	16#00000FE6:
		F_EtherCAT_VendorIDtoString := 'Specter Aerospace Inc.';

	16#00000FE7:
		F_EtherCAT_VendorIDtoString := 'VITZRO VM CO., LTD.';

	16#00000FE8:
		F_EtherCAT_VendorIDtoString := 'Follow Cam Solutions';

	16#00000FE9:
		F_EtherCAT_VendorIDtoString := 'Chengdu Jixing Plasma Technology Co., Ltd.';

	16#00000FEA:
		F_EtherCAT_VendorIDtoString := 'Shenzhen WisdaTech Co., Ltd.';

	16#00000FEC:
		F_EtherCAT_VendorIDtoString := 'Li-tech AS';

	16#00000FED:
		F_EtherCAT_VendorIDtoString := 'Contour Advanced Systems BV';

	16#00000FEE:
		F_EtherCAT_VendorIDtoString := 'Camera Positioning Systems Inc';

	16#00000FEF:
		F_EtherCAT_VendorIDtoString := 'MISUMI (CHINA) PRECISION MACHINERY TRADING CO., LTD.';

	16#00000FF0:
		F_EtherCAT_VendorIDtoString := 'D-CLUE Technologies Co., Ltd.';

	16#00000FF1:
		F_EtherCAT_VendorIDtoString := 'The Board of Trustees of the University of Illinois on behalf of the University of Illinois Chicago';

	16#00000FF2:
		F_EtherCAT_VendorIDtoString := 'Texas A&M University, College of Engineering, J. Mike Walker 66 Department of Mechanical Engineering, Robotics and Automation Design Lab';

	16#00000FF3:
		F_EtherCAT_VendorIDtoString := 'Japan Minicomputer Systems Co., Ltd.';

	16#00000FF4:
		F_EtherCAT_VendorIDtoString := 'Sun Automation Co.,Ltd';

	16#00000FF5:
		F_EtherCAT_VendorIDtoString := 'Puruvesi Automation Inc.';

	16#00000FF6:
		F_EtherCAT_VendorIDtoString := 'Shenzhen Hans Focus Technology Co., Ltd.';

	16#00000FF8:
		F_EtherCAT_VendorIDtoString := 'TAIWAN CHELIC Co., Ltd.';

	16#00000FF9:
		F_EtherCAT_VendorIDtoString := 'RoboDesign Co.,Ltd.';

	16#00000FFA:
		F_EtherCAT_VendorIDtoString := 'PineSolution Co., Ltd.';

	16#00000FFB:
		F_EtherCAT_VendorIDtoString := 'Hangzhou Fisun Intelligency & Technology Co., Ltd.';

	16#00000FFC:
		F_EtherCAT_VendorIDtoString := 'A&D Technology, Inc.';

	16#00000FFD:
		F_EtherCAT_VendorIDtoString := 'IDEC CORPORATION';

	16#00000FFE:
		F_EtherCAT_VendorIDtoString := 'Atel Corp.';

	16#00000FFF:
		F_EtherCAT_VendorIDtoString := 'ZEROSYSTEM CO,LTD';

	16#00001000:
		F_EtherCAT_VendorIDtoString := 'Motiv Robotics, Inc.';

	16#00001001:
		F_EtherCAT_VendorIDtoString := 'Ray-Links (Beijing) Technologies Co., Ltd.';

	16#00001002:
		F_EtherCAT_VendorIDtoString := 'Centro de Automatica y Robotica UPM-CSIC';

	16#00001003:
		F_EtherCAT_VendorIDtoString := 'PLAYTG Co., Ltd.';

	16#00001004:
		F_EtherCAT_VendorIDtoString := 'Shenzhen Huaxin Semiconductor Equipment Technology Co., Ltd.';

	16#00001005:
		F_EtherCAT_VendorIDtoString := 'LT Global Trade Limited dba Eco-Drive Max';

	16#00001006:
		F_EtherCAT_VendorIDtoString := 'SiGaN AG';

	16#00001007:
		F_EtherCAT_VendorIDtoString := 'MOTOREVO ROBOTICS CO.,LTD.';

	16#00001008:
		F_EtherCAT_VendorIDtoString := 'Rheinmetall Canada Inc.';

	16#00001009:
		F_EtherCAT_VendorIDtoString := 'Smart Buildings BVBA';

	16#0000100A:
		F_EtherCAT_VendorIDtoString := 'AixControl GmbH';

	16#0000100B:
		F_EtherCAT_VendorIDtoString := 'Lumina Power, Inc.';

	16#0000100C:
		F_EtherCAT_VendorIDtoString := 'Cryosol-World bv';

	16#0000100D:
		F_EtherCAT_VendorIDtoString := 'Aitoly Instruments Co., Ltd';

	16#0000100E:
		F_EtherCAT_VendorIDtoString := 'FUTUREWORKS';

	16#0000100F:
		F_EtherCAT_VendorIDtoString := 'Changsha University of Science & Technology, School of Physics & Electronic Science';

	16#00001010:
		F_EtherCAT_VendorIDtoString := 'NEXTW Technology CO., LTD.';

	16#00001011:
		F_EtherCAT_VendorIDtoString := 'H4 Inc.';

	16#00001012:
		F_EtherCAT_VendorIDtoString := 'ZHEJIANG SUPCON INFORMATION CO.,LTD.';

	16#00001013:
		F_EtherCAT_VendorIDtoString := 'oKSitem Otomasyon Ltd. Sti.';

	16#00001014:
		F_EtherCAT_VendorIDtoString := 'CSIM INC.';

	16#00001015:
		F_EtherCAT_VendorIDtoString := 'Valvan NV';

	16#00001016:
		F_EtherCAT_VendorIDtoString := 'ASAHI ENGINEERING CO.,LTD.';

	16#00001017:
		F_EtherCAT_VendorIDtoString := 'Weifang Ouxin Intelligent Control Technology Co., LTD';

	16#00001018:
		F_EtherCAT_VendorIDtoString := 'GZ Photonics Technology Co., Ltd.';

	16#00001019:
		F_EtherCAT_VendorIDtoString := 'Optoscan S.r.l.';

	16#0000101A:
		F_EtherCAT_VendorIDtoString := 'Ningbo Huayuan Machinery Technology Co., Ltd.';

	16#0000101B:
		F_EtherCAT_VendorIDtoString := 'Laza Medical, Inc.';

	16#0000101C:
		F_EtherCAT_VendorIDtoString := 'Vectioneer BV';

	16#0000101D:
		F_EtherCAT_VendorIDtoString := 'Huasteigen (Ningbo) Automation Technology Co.,Ltd.';

	16#00001020:
		F_EtherCAT_VendorIDtoString := 'PDM Industrial Excellence B.V.';

	16#00001022:
		F_EtherCAT_VendorIDtoString := 'SV Sistemi di Sicurezza';

	16#00001023:
		F_EtherCAT_VendorIDtoString := 'Lynx Robotics LLC';

	16#00001024:
		F_EtherCAT_VendorIDtoString := 'Jcast Networks Korea, Inc.';

	16#00001025:
		F_EtherCAT_VendorIDtoString := 'AcroComm Corporation';

	16#00001026:
		F_EtherCAT_VendorIDtoString := 'Hacint Intelligence Technology Co., Ltd.';

	16#00001027:
		F_EtherCAT_VendorIDtoString := 'Vision Hardware Partner';

	16#00001028:
		F_EtherCAT_VendorIDtoString := 'Forbes Marshall Pvt. Ltd.';

	16#00001029:
		F_EtherCAT_VendorIDtoString := 'Shenzhen Sunvision Technology Co., Ltd.';

	16#0000102A:
		F_EtherCAT_VendorIDtoString := 'ASAP Electronics GmbH';

	16#0000102B:
		F_EtherCAT_VendorIDtoString := 'Matrox Electronic Systems Ltd.';

	16#0000102C:
		F_EtherCAT_VendorIDtoString := 'Shanghai Zhentai Instrument Co., Ltd.';

	16#0000102D:
		F_EtherCAT_VendorIDtoString := 'ROHM Co., Ltd.';

	16#0000102E:
		F_EtherCAT_VendorIDtoString := 'Chengdu SeaDee Technology Co.,Ltd.';

	16#0000102F:
		F_EtherCAT_VendorIDtoString := 'Huazhuo Measurement and Control Technology (Shenzhen) Co., Ltd.';

	16#00001030:
		F_EtherCAT_VendorIDtoString := 'Advanced Design Technology Co.,Ltd';

	16#00001031:
		F_EtherCAT_VendorIDtoString := 'MI-Partners B.V.';

	16#00001032:
		F_EtherCAT_VendorIDtoString := 'Beijing Hanwen Wangxing Technology Co., Ltd';

	16#00001033:
		F_EtherCAT_VendorIDtoString := 'nexo SrL';

	16#00001034:
		F_EtherCAT_VendorIDtoString := 'Simplex Motion AB';

	16#00001035:
		F_EtherCAT_VendorIDtoString := 'Wuxi Juxie Intelligent Drive Co.,Ltd.';

	16#00001036:
		F_EtherCAT_VendorIDtoString := 'Shenzhen Huizhong Intelligent Technology Co., Ltd';

	16#00001037:
		F_EtherCAT_VendorIDtoString := 'THEISSL systems GmbH';

	16#00001038:
		F_EtherCAT_VendorIDtoString := 'VOLAS GmbH';

	16#00001039:
		F_EtherCAT_VendorIDtoString := 'ASTI Corporation';

	16#0000103A:
		F_EtherCAT_VendorIDtoString := 'ELETTRONICA G.B. SRL';

	16#0000103B:
		F_EtherCAT_VendorIDtoString := 'VELTRU AG';

	16#0000103C:
		F_EtherCAT_VendorIDtoString := 'SEMISOL Co., Ltd.';

	16#0000103D:
		F_EtherCAT_VendorIDtoString := 'GENIWORX Co., Ltd.';

	16#0000103E:
		F_EtherCAT_VendorIDtoString := 'TUODAO (SINGAPORE) PTE. LTD.';

	16#00001041:
		F_EtherCAT_VendorIDtoString := 'SISGEO SRL';

	16#00001043:
		F_EtherCAT_VendorIDtoString := 'Oelmaier Automation GmbH';

	16#00001044:
		F_EtherCAT_VendorIDtoString := 'VISHAY ADVANCED TECHNOLOGIES LTD';

	16#00001045:
		F_EtherCAT_VendorIDtoString := 'Beyond Kinematics LLC';

	16#00001046:
		F_EtherCAT_VendorIDtoString := 'Control expertise for trading Co. LTD';

	16#00001047:
		F_EtherCAT_VendorIDtoString := 'Tujian Automation Technology (Suzhou) Co., Ltd.';

	16#00001048:
		F_EtherCAT_VendorIDtoString := 'Shibaura Machine Co., Ltd.';

	16#00001049:
		F_EtherCAT_VendorIDtoString := 'Chip Right Corporation';

	16#0000104A:
		F_EtherCAT_VendorIDtoString := 'American Superconductor Corporation';

	16#0000104B:
		F_EtherCAT_VendorIDtoString := 'Emirates Automation Pvt Ltd';

	16#0000104C:
		F_EtherCAT_VendorIDtoString := 'ERL Sensors and Automation';

	16#0000104D:
		F_EtherCAT_VendorIDtoString := 'Zhuhai Yuanshicheng Technology Co., Ltd.';

	16#0000104E:
		F_EtherCAT_VendorIDtoString := 'University of Bergamo, Department of Engineering and Applied Sciences, Mechatronics and Mechanical Dynamics Lab';

	16#0000104F:
		F_EtherCAT_VendorIDtoString := 'Maxell Frontier Co., Ltd.';

	16#00001050:
		F_EtherCAT_VendorIDtoString := 'ZENSTEM CO., LTD.';

	16#00001051:
		F_EtherCAT_VendorIDtoString := 'CONEC Elektronische Bauelemente GmbH';

	16#00001052:
		F_EtherCAT_VendorIDtoString := 'Teegarden Engineering S.r.l.';

	16#00001053:
		F_EtherCAT_VendorIDtoString := 'iFORCOM KYOEI Co., Ltd.';

	16#00001054:
		F_EtherCAT_VendorIDtoString := 'Timeback Inc. dba Reflex Robotics';

	16#00001055:
		F_EtherCAT_VendorIDtoString := 'Stryker Corporation';

	16#00001056:
		F_EtherCAT_VendorIDtoString := 'Kickmaker';

	16#00001057:
		F_EtherCAT_VendorIDtoString := 'Andar Elektromekanik Sistemler Sanayi ve Ticaret Anonim Şirketi';

	16#00001058:
		F_EtherCAT_VendorIDtoString := 'Hefei Kaiyue Semiconductor Technology Co., Ltd.';

	16#00001059:
		F_EtherCAT_VendorIDtoString := 'Clean-Lasersysteme GmbH';

	16#0000105A:
		F_EtherCAT_VendorIDtoString := 'SMACH CO., Ltd.';

	16#0000105B:
		F_EtherCAT_VendorIDtoString := 'ACD Elektronik GmbH';

	16#0000105C:
		F_EtherCAT_VendorIDtoString := 'Jiangsu Houjing Technology Co., Ltd.';

	16#0000105D:
		F_EtherCAT_VendorIDtoString := 'TACSCO Co., Ltd';

	16#0000105E:
		F_EtherCAT_VendorIDtoString := 'DGA Maitrise de linformation';

	16#0000105F:
		F_EtherCAT_VendorIDtoString := 'Dasstec B2B SRL';

	16#00001060:
		F_EtherCAT_VendorIDtoString := 'Comau S.p.A.';

	16#00001061:
		F_EtherCAT_VendorIDtoString := 'Vertiv Group Corporation';

	16#00001062:
		F_EtherCAT_VendorIDtoString := 'Insystems Inc.';

	16#00001063:
		F_EtherCAT_VendorIDtoString := 'Digital Sports Solutions LLC';

	16#00001064:
		F_EtherCAT_VendorIDtoString := 'BorgRoid Inc.';

	16#00001066:
		F_EtherCAT_VendorIDtoString := 'Shanghai ZeroOne Information Technology Co., Ltd.';

	16#00001067:
		F_EtherCAT_VendorIDtoString := 'STREAK – Engenharia em Automacao, LDA';

	16#00001068:
		F_EtherCAT_VendorIDtoString := 'Seurat Technologies, Inc.';

	16#00001069:
		F_EtherCAT_VendorIDtoString := 'EMBETTER TECHNOLOGIES PRIVATE LIMITED';

	16#0000106A:
		F_EtherCAT_VendorIDtoString := 'Beijing Regulate Technology Co., Ltd.';

	16#0000106B:
		F_EtherCAT_VendorIDtoString := 'Electronics Corporation of India Ltd.';

	16#0000106C:
		F_EtherCAT_VendorIDtoString := 'Cargt, Inc';

	16#0000106D:
		F_EtherCAT_VendorIDtoString := 'Shanghai Paipin Optoelectronic Technology Co., Ltd.';

	16#0000106E:
		F_EtherCAT_VendorIDtoString := 'Coherent Switzerland AG';

	16#0000106F:
		F_EtherCAT_VendorIDtoString := 'IP CAMP Limited Liability Company';

	16#00001071:
		F_EtherCAT_VendorIDtoString := 'Suzhou Ouluda Intelligent Technology Co., Ltd.';

	16#00001073:
		F_EtherCAT_VendorIDtoString := 'K&S Advanced Systems LTD';

	16#00001074:
		F_EtherCAT_VendorIDtoString := 'Roche Diagnostics GmbH';

	16#00001075:
		F_EtherCAT_VendorIDtoString := 'FerRobotics Compliant Robot Technology GmbH';

	16#00001077:
		F_EtherCAT_VendorIDtoString := 'TOKY ELECTRICAL CO., LTD.';

	16#00001078:
		F_EtherCAT_VendorIDtoString := 'ET Systems Engineering d.o.o.';

	16#00001079:
		F_EtherCAT_VendorIDtoString := 'Electrovia Technologies Corp';

	16#0000107A:
		F_EtherCAT_VendorIDtoString := 'Imperix Ltd.';

	16#0000107B:
		F_EtherCAT_VendorIDtoString := 'FoodJet B.V.';

	16#0000107C:
		F_EtherCAT_VendorIDtoString := 'Meridian Laboratory, Inc.';

	16#0000107D:
		F_EtherCAT_VendorIDtoString := 'ITECH ELECTRONIC CO., LTD.';

	16#0000107E:
		F_EtherCAT_VendorIDtoString := 'DANNIE ELEKTRONİK VE ELEKTRİK LTD.';

	16#0000107F:
		F_EtherCAT_VendorIDtoString := 'logi.cals GmbH';

	16#00001080:
		F_EtherCAT_VendorIDtoString := 'Unionx (Wuhan) Industrial Technology Co., Ltd.';

	16#00001081:
		F_EtherCAT_VendorIDtoString := 'Shenzhen ASunDar Electronics Co., Ltd.';

	16#00001082:
		F_EtherCAT_VendorIDtoString := 'Artesyn Embedded Technologies Philippines Inc.';

	16#00001083:
		F_EtherCAT_VendorIDtoString := 'Wuxi Dixin Technology Co., Ltd.';

	16#00001084:
		F_EtherCAT_VendorIDtoString := 'Philips Health Technology (China) Co., Ltd Suzhou Branch';

	16#00001085:
		F_EtherCAT_VendorIDtoString := 'Zhuzhou Jiacheng Science & Technology Development Co., Ltd.';

	16#00001086:
		F_EtherCAT_VendorIDtoString := 'Tinius Olsen Testing Machine Company';

	16#00001087:
		F_EtherCAT_VendorIDtoString := 'Mettler-Toledo (Changzhou) Measurement Technology Ltd.';

	16#00001088:
		F_EtherCAT_VendorIDtoString := 'Vermes Microdispensing GmbH';

	16#00001089:
		F_EtherCAT_VendorIDtoString := 'ASDEA HARDWARE SRL';

	16#0000108A:
		F_EtherCAT_VendorIDtoString := 'GE Vernova Advanced Research';

	16#0000108B:
		F_EtherCAT_VendorIDtoString := 'Nanjing Estun Codroid Technology Co.,Ltd.';

	16#0000108C:
		F_EtherCAT_VendorIDtoString := 'Reilhofer KG';

	16#0000108D:
		F_EtherCAT_VendorIDtoString := 'Shenzhen accurate measurement and processing Technology Co Ltd';

	16#0000108E:
		F_EtherCAT_VendorIDtoString := 'AWL-Techniek B.V.';

	16#0000108F:
		F_EtherCAT_VendorIDtoString := 'IDEM Safety Switches Ltd.';

	16#00001090:
		F_EtherCAT_VendorIDtoString := 'SHANGHAI TOSUN Technology Ltd.';

	16#00001091:
		F_EtherCAT_VendorIDtoString := 'ITBB Institut fur Technologien der Biomechanik und Biomaterialien GmbH';

	16#00001093:
		F_EtherCAT_VendorIDtoString := 'SSP Safety System Products GmbH & Co. KG';

	16#00001094:
		F_EtherCAT_VendorIDtoString := 'Linx Global Mfg., LLC';

	16#000010FA:
		F_EtherCAT_VendorIDtoString := 'Beijing BBF Servo Technology Co.,Ltd.';

	16#00001101:
		F_EtherCAT_VendorIDtoString := 'Suzhou BOE Sensor Technology Co., Ltd.';

	16#00001110:
		F_EtherCAT_VendorIDtoString := 'A-KYUNG Motion Inc.';

	16#00001111:
		F_EtherCAT_VendorIDtoString := 'MLS Lanny GmbH';

	16#00001119:
		F_EtherCAT_VendorIDtoString := 'Mettler-Toledo GmbH';

	16#00001122:
		F_EtherCAT_VendorIDtoString := 'CanTops';

	16#00001132:
		F_EtherCAT_VendorIDtoString := 'FERAG AG';

	16#0000115C:
		F_EtherCAT_VendorIDtoString := 'YASKAWA Europe GmbH';

	16#0000115F:
		F_EtherCAT_VendorIDtoString := 'K-TRONIC S.r.l';

	16#00001186:
		F_EtherCAT_VendorIDtoString := 'Ching Tai Electric Wire & Cable Co., Ltd.';

	16#00001191:
		F_EtherCAT_VendorIDtoString := 'Techno Create, Inc.';

	16#00001204:
		F_EtherCAT_VendorIDtoString := 'EAST Group Co., Ltd.';

	16#00001219:
		F_EtherCAT_VendorIDtoString := 'Contexa SA';

	16#00001298:
		F_EtherCAT_VendorIDtoString := 'Shenzhen Honestar Electronics Co., Ltd';

	16#000012A5:
		F_EtherCAT_VendorIDtoString := 'i2A Systems Co., Ltd.';

	16#000012AD:
		F_EtherCAT_VendorIDtoString := 'VIVAVIS AG';

	16#0000130C:
		F_EtherCAT_VendorIDtoString := 'MotionTech AS';

	16#00001314:
		F_EtherCAT_VendorIDtoString := 'Beijing Art Technology Development Co., Ltd.';

	16#00001337:
		F_EtherCAT_VendorIDtoString := 'rt-labs AB';

	16#00001357:
		F_EtherCAT_VendorIDtoString := 'Cosmo Instruments Co.,Ltd.';

	16#000013FE:
		F_EtherCAT_VendorIDtoString := 'Advantech Co., Ltd.';

	16#00001430:
		F_EtherCAT_VendorIDtoString := 'ChengDu HiCNC Equipment Co., Ltd.';

	16#0000144A:
		F_EtherCAT_VendorIDtoString := 'ADLINK TECHNOLOGY INC.';

	16#0000147A:
		F_EtherCAT_VendorIDtoString := 'eubus GmbH';

	16#000014FF:
		F_EtherCAT_VendorIDtoString := 'Precise Automation, Inc.';

	16#00001502:
		F_EtherCAT_VendorIDtoString := 'Unico Inc.';

	16#0000150E:
		F_EtherCAT_VendorIDtoString := 'Ono Sokki Co. Ltd.';

	16#00001521:
		F_EtherCAT_VendorIDtoString := 'CHIKO AIRTEC CO., LTD.';

	16#00001525:
		F_EtherCAT_VendorIDtoString := 'Newson NV';

	16#00001582:
		F_EtherCAT_VendorIDtoString := 'TRsystems GmbH';

	16#00001600:
		F_EtherCAT_VendorIDtoString := 'Helmholtz-Zentrum Dresden-Rossendorf e.V.';

	16#00001616:
		F_EtherCAT_VendorIDtoString := 'DLR Deutsches Zentrum fur Luft- und Raumfahrt e.V.';

	16#00001619:
		F_EtherCAT_VendorIDtoString := 'Kyoto Denkiki Co.,Ltd.';

	16#00001666:
		F_EtherCAT_VendorIDtoString := 'Shenzhen Softwin Technology Co., LTD';

	16#0000166D:
		F_EtherCAT_VendorIDtoString := 'YXLON International GmbH';

	16#00001688:
		F_EtherCAT_VendorIDtoString := 'Shanghai Allinmodule Intelligence Co., Ltd';

	16#00001701:
		F_EtherCAT_VendorIDtoString := 'PLR Pruftechnik Linke & Ruhe GmbH';

	16#00001729:
		F_EtherCAT_VendorIDtoString := 'Shibaura Machine India Private Limited';

	16#0000177A:
		F_EtherCAT_VendorIDtoString := 'NanJing Aegis-Iron Technology Co., Ltd.';

	16#00001783:
		F_EtherCAT_VendorIDtoString := 'Inaba Denki Sangyo Co., Ltd.';

	16#00001799:
		F_EtherCAT_VendorIDtoString := 'K-one Co., Ltd.';

	16#0000179A:
		F_EtherCAT_VendorIDtoString := 'HEIG-VD - Haute Ecole dIngenierie et de Gestion du Canton de Vaud';

	16#00001800:
		F_EtherCAT_VendorIDtoString := 'TAMAGAWA SEIKI CO.,LTD.';

	16#00001809:
		F_EtherCAT_VendorIDtoString := 'LLC DOMINANTA-STAGE';

	16#00001810:
		F_EtherCAT_VendorIDtoString := 'L & S Electric, Inc.';

	16#00001818:
		F_EtherCAT_VendorIDtoString := 'Fujian Huafeng New Materials Co. Ltd.';

	16#00001848:
		F_EtherCAT_VendorIDtoString := 'Keysight Technologies Deutschland GmbH';

	16#00001895:
		F_EtherCAT_VendorIDtoString := 'HOERBIGER Wien GmbH';

	16#00001899:
		F_EtherCAT_VendorIDtoString := 'Hagenuk Marinekommunikation GmbH';

	16#00001919:
		F_EtherCAT_VendorIDtoString := 'SACMI IMOLA S.C.';

	16#00001946:
		F_EtherCAT_VendorIDtoString := 'AMADA Co., Ltd.';

	16#00001962:
		F_EtherCAT_VendorIDtoString := 'Tomsk State University of Control Systems and Radioelectronics, Institute of Innovations';

	16#00001980:
		F_EtherCAT_VendorIDtoString := 'HANMI Semiconductor Co., Ltd.';

	16#00001984:
		F_EtherCAT_VendorIDtoString := 'LAUMAS Elettronica s.r.l.';

	16#00001987:
		F_EtherCAT_VendorIDtoString := 'DINA Elektronik GmbH';

	16#00001991:
		F_EtherCAT_VendorIDtoString := 'Shenzhen Samkoon Technology Co., Ltd.';

	16#00001993:
		F_EtherCAT_VendorIDtoString := 'PushCorp, Inc.';

	16#00001997:
		F_EtherCAT_VendorIDtoString := 'MEDICAL TECHNOLOGIES Ltd';

	16#00001A05:
		F_EtherCAT_VendorIDtoString := 'SYN-TEK Automation Co., Ltd.';

	16#00001A1D:
		F_EtherCAT_VendorIDtoString := 'Guangdong Ruobo Intelligent Robot Co., Ltd.';

	16#00001A21:
		F_EtherCAT_VendorIDtoString := 'BySTORM & CO. srl';

	16#00001A85:
		F_EtherCAT_VendorIDtoString := 'Michel Van de Wiele NV';

	16#00001A90:
		F_EtherCAT_VendorIDtoString := 'IPETRONIK GmbH & Co. KG';

	16#00001B2C:
		F_EtherCAT_VendorIDtoString := 'Opal-RT Technologies, Inc.';

	16#00001B66:
		F_EtherCAT_VendorIDtoString := 'Sennheiser electronic GmbH & Co. KG';

	16#00001BCB:
		F_EtherCAT_VendorIDtoString := 'Bustec Ltd.';

	16#00001C80:
		F_EtherCAT_VendorIDtoString := 'Hoffmann + Krippner GmbH';

	16#00001DFC:
		F_EtherCAT_VendorIDtoString := 'Shaanxi Yidu Intelligent Technology Co., Ltd.';

	16#00001E8A:
		F_EtherCAT_VendorIDtoString := 'Esima Endustriyel ve Elektronik Sistemler San. ve Tic. Ltd. Şti';

	16#00002000:
		F_EtherCAT_VendorIDtoString := 'Motiv Space Systems, Inc.';

	16#00002001:
		F_EtherCAT_VendorIDtoString := 'Nextec Technologies 2001 Ltd.';

	16#00002010:
		F_EtherCAT_VendorIDtoString := 'Shenzhen Xhorse Electronics Co., Ltd.';

	16#00002014:
		F_EtherCAT_VendorIDtoString := 'Capcon (Guangdong-Macao In-Depth Cooperation Zone) Co., Ltd';

	16#00002015:
		F_EtherCAT_VendorIDtoString := 'GW (Shanghai) Laser Technology Co., Ltd.';

	16#00002018:
		F_EtherCAT_VendorIDtoString := 'Thermo Fisher Scientific (Bremen) GmbH';

	16#00002019:
		F_EtherCAT_VendorIDtoString := 'Komito Bleu BVBA';

	16#00002020:
		F_EtherCAT_VendorIDtoString := 'NanJing KaiTong Automation Technology Co., Ltd.';

	16#00002021:
		F_EtherCAT_VendorIDtoString := 'Wuhan Lorenz Technology Co., Ltd.';

	16#000021DE:
		F_EtherCAT_VendorIDtoString := 'Ruthi Electronic AG';

	16#00002055:
		F_EtherCAT_VendorIDtoString := 'Bristol Robotics Laboratory';

	16#0000205E:
		F_EtherCAT_VendorIDtoString := 'HyVISION SYSTEM Inc.';

	16#00002103:
		F_EtherCAT_VendorIDtoString := 'ASE Co., Ltd.';

	16#00002186:
		F_EtherCAT_VendorIDtoString := 'Sobal Corporation';

	16#000021C1:
		F_EtherCAT_VendorIDtoString := 'ATSENSE INC.';

	16#000022CD:
		F_EtherCAT_VendorIDtoString := 'Kinova Inc.';

	16#000022D2:
		F_EtherCAT_VendorIDtoString := 'Synapticon GmbH';

	16#00002304:
		F_EtherCAT_VendorIDtoString := 'DANIELI AUTOMATION SPA';

	16#00002380:
		F_EtherCAT_VendorIDtoString := 'Nanjing SCIYON Automation Group Co., Ltd.';

	16#00002400:
		F_EtherCAT_VendorIDtoString := 'Daikoku Innovations LLP';

	16#00002501:
		F_EtherCAT_VendorIDtoString := 'EO Technics Co., Ltd.';

	16#00002518:
		F_EtherCAT_VendorIDtoString := 'KUBO Technologies LLC';

	16#00002631:
		F_EtherCAT_VendorIDtoString := 'MICROPAP ENGINEERING SL';

	16#0000266D:
		F_EtherCAT_VendorIDtoString := 'Comet AG';

	16#00002727:
		F_EtherCAT_VendorIDtoString := 'Altra Industrial Motion do Brasil Equipamentos Industriais LTDA';

	16#0000276A:
		F_EtherCAT_VendorIDtoString := 'Shenzhen SuperFar lntelligent Control Technology Co.,LTD.';

	16#000027AB:
		F_EtherCAT_VendorIDtoString := 'Rollmann Elektronik';

	16#00002838:
		F_EtherCAT_VendorIDtoString := 'burster prazisionsmesstechnik gmbh & co kg';

	16#00002888:
		F_EtherCAT_VendorIDtoString := 'TCOS System Sdn Bhd';

	16#00002910:
		F_EtherCAT_VendorIDtoString := 'Shenzhen Yishu Technology Co., Ltd.';

	16#00002939:
		F_EtherCAT_VendorIDtoString := 'Zaber Technologies Inc.';

	16#00002A3F:
		F_EtherCAT_VendorIDtoString := 'Shenzhen RUI Intelligent Control Co.,Ltd.';

	16#00002AA8:
		F_EtherCAT_VendorIDtoString := 'NiniX Technologies NV';

	16#00002CE7:
		F_EtherCAT_VendorIDtoString := 'NiLAB GmbH';

	16#00002ECC:
		F_EtherCAT_VendorIDtoString := 'PSK Inc.';

	16#000030E0:
		F_EtherCAT_VendorIDtoString := 'DotLine GmbH';

	16#00003181:
		F_EtherCAT_VendorIDtoString := 'HaptX Inc.';

	16#000031CF:
		F_EtherCAT_VendorIDtoString := 'Schleiheimer Soft- und Hardwareentwicklung GmbH';

	16#00003333:
		F_EtherCAT_VendorIDtoString := 'Protokit Robotics Pty Ltd';

	16#00003388:
		F_EtherCAT_VendorIDtoString := 'MEIJI ELECTRIC INDUSTRIES CO., LTD.';

	16#000033AA:
		F_EtherCAT_VendorIDtoString := 'Sanlab Yazilim Arastirma Gelistirme Enerji Muhendislik San. ve Tic. Ltd. Sti';

	16#000033C3:
		F_EtherCAT_VendorIDtoString := 'MatrixGroup (CMS) Pty Ltd';

	16#00003443:
		F_EtherCAT_VendorIDtoString := '4C Electronics Limited';

	16#00003456:
		F_EtherCAT_VendorIDtoString := 'Guangzhou Automobile Group Co., Ltd. Automotive Engineering Research and Development Center';

	16#00003508:
		F_EtherCAT_VendorIDtoString := 'PURPOSE CO., LTD';

	16#00003535:
		F_EtherCAT_VendorIDtoString := 'ASAHI ENTERPRISE';

	16#00003610:
		F_EtherCAT_VendorIDtoString := 'eProLinkTek Co., Ltd.';

	16#00003777:
		F_EtherCAT_VendorIDtoString := 'UBI, Inc.';

	16#00003853:
		F_EtherCAT_VendorIDtoString := 'Shenzhen ICM Technology Development Co.,Ltd.';

	16#00004000:
		F_EtherCAT_VendorIDtoString := 'Automotive Parts and Accessory Systems (APAS) R&D Centre';

	16#00004100:
		F_EtherCAT_VendorIDtoString := 'Fusion Information Technology Co., Ltd.';

	16#00004123:
		F_EtherCAT_VendorIDtoString := 'University of Basel, Faculty of Medicine';

	16#0000414C:
		F_EtherCAT_VendorIDtoString := 'ALIARO AB';

	16#00004150:
		F_EtherCAT_VendorIDtoString := 'Korea Advanced Institute of Science and Technology, College of Engineering, Department of Mechanical Engineering, Robotics & Artificial Intelligence Lab';

	16#00004154:
		F_EtherCAT_VendorIDtoString := 'acontis technologies GmbH';

	16#000041EC:
		F_EtherCAT_VendorIDtoString := 'Interactive Engineering Corporation';

	16#000042AB:
		F_EtherCAT_VendorIDtoString := 'Andi Packaging Technology (Guangdong) Co., Ltd.';

	16#00004301:
		F_EtherCAT_VendorIDtoString := 'Ocean Optics, Inc.';

	16#00004305:
		F_EtherCAT_VendorIDtoString := 'Order One Solutions, LLC';

	16#00004321:
		F_EtherCAT_VendorIDtoString := 'Leadshine Technology Co., Ltd.';

	16#0000434C:
		F_EtherCAT_VendorIDtoString := 'CIRCLE LAB';

	16#0000434D:
		F_EtherCAT_VendorIDtoString := 'Columbus McKinnon Corporation';

	16#00004351:
		F_EtherCAT_VendorIDtoString := 'OPCsoft Co., Ltd.';

	16#00004369:
		F_EtherCAT_VendorIDtoString := 'SHYANG BAO INC.';

	16#00004441:
		F_EtherCAT_VendorIDtoString := 'Myostat Motion Control Inc.';

	16#0000444E:
		F_EtherCAT_VendorIDtoString := 'DN Solutions Co., Ltd.';

	16#00004468:
		F_EtherCAT_VendorIDtoString := 'Jiangsu Zhongxinke Technology Co.,Ltd.';

	16#00004553:
		F_EtherCAT_VendorIDtoString := 'Energy Support Corporation';

	16#00004567:
		F_EtherCAT_VendorIDtoString := 'Shanghai University';

	16#00004604:
		F_EtherCAT_VendorIDtoString := 'Budker Institute of Nuclear Physics of Siberian Branch Russian Academy of Sciences (BINP SB RAS)';

	16#00004654:
		F_EtherCAT_VendorIDtoString := 'FUKOKU TOKAI Co., Ltd.';

	16#00004685:
		F_EtherCAT_VendorIDtoString := 'Sandensha Co., Ltd.';

	16#00004711:
		F_EtherCAT_VendorIDtoString := 'FRABA B.V.';

	16#00004717:
		F_EtherCAT_VendorIDtoString := 'Hanwha Ocean Co., Ltd.';

	16#00004752:
		F_EtherCAT_VendorIDtoString := 'Generic Robotics Limited';

	16#00004845:
		F_EtherCAT_VendorIDtoString := 'Haller + Erne GmbH';

	16#00004943:
		F_EtherCAT_VendorIDtoString := 'INTER CONTROL Hermann Kohler Elektrik GmbH & Co. KG';

	16#00004957:
		F_EtherCAT_VendorIDtoString := 'INTERWORKS Co., Ltd.';

	16#00004B41:
		F_EtherCAT_VendorIDtoString := 'Kratzer Automation AG';

	16#00004D43:
		F_EtherCAT_VendorIDtoString := 'SKS Control OY';

	16#00004D50:
		F_EtherCAT_VendorIDtoString := 'Max-Planck-Institut fur extraterestrische Physik';

	16#00004D63:
		F_EtherCAT_VendorIDtoString := 'MAGICS Instruments NV';

	16#00004E01:
		F_EtherCAT_VendorIDtoString := 'REON Technology, Inc.';

	16#00005050:
		F_EtherCAT_VendorIDtoString := 'TSUZUKI DENKI CO., LTD';

	16#00005052:
		F_EtherCAT_VendorIDtoString := 'Proekspert AS';

	16#00005053:
		F_EtherCAT_VendorIDtoString := 'PRESTOSOLUTION Ltd.';

	16#00005071:
		F_EtherCAT_VendorIDtoString := 'COTS Technology Co., Ltd.';

	16#00005100:
		F_EtherCAT_VendorIDtoString := 'WOORI Technology Inc.';

	16#00005146:
		F_EtherCAT_VendorIDtoString := 'Ningbo Qifan Automation Technology Co., LTD';

	16#00005244:
		F_EtherCAT_VendorIDtoString := 'Desird Tasarim Arge Uygulama Elektronik Destek Ithalat Ihracat San. ve Tic. Ltd. Sti.';

	16#00005257:
		F_EtherCAT_VendorIDtoString := 'Rosch & Walter Industrie-Elektronik GmbH';

	16#00005341:
		F_EtherCAT_VendorIDtoString := 'SOHOAID Corporation';

	16#00005368:
		F_EtherCAT_VendorIDtoString := 'WUHAN SHARE AUTOMATION TECHNOLOGY CO.,LTD';

	16#00005493:
		F_EtherCAT_VendorIDtoString := 'Sanlien Technology Corp.';

	16#00005549:
		F_EtherCAT_VendorIDtoString := 'Genius Technology Co., Ltd.';

	16#00005858:
		F_EtherCAT_VendorIDtoString := 'Shenyang REDTECH Electric Co., Ltd.';

	16#00005995:
		F_EtherCAT_VendorIDtoString := 'Kristl, Seibt & Co GmbH';

	16#00005F0A:
		F_EtherCAT_VendorIDtoString := 'Technische Universitat Darmstadt, Fachgebiet Elektrotechnik und Informationstechnik';

	16#00005F5F:
		F_EtherCAT_VendorIDtoString := 'Maurizio Ferraris (dba Studio Ferraris)';

	16#00006001:
		F_EtherCAT_VendorIDtoString := 'Shanghai HiFound Control Electronic Technology Co., Ltd';

	16#00006084:
		F_EtherCAT_VendorIDtoString := 'Gerber Technology Inc.';

	16#000060C8:
		F_EtherCAT_VendorIDtoString := 'KUKA Deutschland GmbH';

	16#000060C9:
		F_EtherCAT_VendorIDtoString := 'KUKA Robotics China Co., Ltd.';

	16#000060CB:
		F_EtherCAT_VendorIDtoString := 'Hitachi Zosen Corporation, Precision Machinery Headquarters, Electronic Control Business Unit';

	16#00006100:
		F_EtherCAT_VendorIDtoString := 'Kurvatur A/S';

	16#00006145:
		F_EtherCAT_VendorIDtoString := 'Shenzhen Huanan Numerical Control System Co., Ltd.';

	16#00006339:
		F_EtherCAT_VendorIDtoString := 'SINTOKOGIO, LTD.';

	16#00006432:
		F_EtherCAT_VendorIDtoString := 'Beijing Jingwei Hirain Technologies Co., Inc.';

	16#00006482:
		F_EtherCAT_VendorIDtoString := 'YUSHIN PRECISION EQUIPMENT CO., LTD.';

	16#00006500:
		F_EtherCAT_VendorIDtoString := 'Triductor Technology(Suzhou), Inc';

	16#00006666:
		F_EtherCAT_VendorIDtoString := 'Qingdao Technological University, College of Mechanical Engineering';

	16#00006688:
		F_EtherCAT_VendorIDtoString := 'Gsolar Power Co., Ltd.';

	16#00006741:
		F_EtherCAT_VendorIDtoString := 'NIPPON SIGNAL CO.,LTD.';

	16#00006789:
		F_EtherCAT_VendorIDtoString := 'University of Electronic Science and Technology of China';

	16#00006888:
		F_EtherCAT_VendorIDtoString := 'Shenzhen Hayhon Equipment Technologies Co., LTD';

	16#00006889:
		F_EtherCAT_VendorIDtoString := 'JKControl Co., Ltd.';

	16#00006A64:
		F_EtherCAT_VendorIDtoString := 'Beijing Jingdiao Co., Ltd.';

	16#00006A6B:
		F_EtherCAT_VendorIDtoString := 'JK Robots Co., Ltd.';

	16#00006C78:
		F_EtherCAT_VendorIDtoString := 'N.A.T. GmbH';

	16#00007071:
		F_EtherCAT_VendorIDtoString := 'Thermal Dynamics Oy';

	16#00007073:
		F_EtherCAT_VendorIDtoString := 'Mahr GmbH';

	16#00007170:
		F_EtherCAT_VendorIDtoString := 'Hyundai Robotics Co., Ltd.';

	16#00007203:
		F_EtherCAT_VendorIDtoString := 'TOYOTA MOTOR CORPORATION';

	16#00007217:
		F_EtherCAT_VendorIDtoString := 'YunKe Intelligent Servo Control Technology Co.,Ltd.';

	16#00007220:
		F_EtherCAT_VendorIDtoString := 'Shenyang Machine Tool(Group) Research & Design Institute Co,Ltd. Shanghai Branch';

	16#00007404:
		F_EtherCAT_VendorIDtoString := 'Veawe Info Dynamics Pvt. Ltd.';

	16#00007595:
		F_EtherCAT_VendorIDtoString := 'LS Mecapion Co., Ltd.';

	16#00007604:
		F_EtherCAT_VendorIDtoString := 'ONTEC CO., LTD';

	16#00007680:
		F_EtherCAT_VendorIDtoString := 'HUNAN SUPER INFORMATION CO., LTD';

	16#00007684:
		F_EtherCAT_VendorIDtoString := 'LOGTICS Inc.';

	16#00007715:
		F_EtherCAT_VendorIDtoString := 'Foxnum Technology Co., Ltd.';

	16#00007716:
		F_EtherCAT_VendorIDtoString := 'Kyoei Electronics Co., Ltd.';

	16#00007777:
		F_EtherCAT_VendorIDtoString := 'Sheltronics Control Systems Private Limited';

	16#00007880:
		F_EtherCAT_VendorIDtoString := 'NISSIN SYSTEMS Co., Ltd.';

	16#00007978:
		F_EtherCAT_VendorIDtoString := 'Junchuang (Xiamen) Automation Technology Co., Ltd.';

	16#00007A17:
		F_EtherCAT_VendorIDtoString := 'Tait Towers Manufacturing, LLC';

	16#00007EC5:
		F_EtherCAT_VendorIDtoString := 'tec5 AG';

	16#00008027:
		F_EtherCAT_VendorIDtoString := 'Tech Mahindra Ltd.';

	16#00008055:
		F_EtherCAT_VendorIDtoString := 'Ethereal Machines Pvt. Ltd.';

	16#00008086:
		F_EtherCAT_VendorIDtoString := 'Intel Corporation';

	16#00008281:
		F_EtherCAT_VendorIDtoString := 'China Electric Power Research Institute (CEPRI)';

	16#00008355:
		F_EtherCAT_VendorIDtoString := 'Hybrid Energy Storage Solutions S.L.';

	16#00008421:
		F_EtherCAT_VendorIDtoString := 'Raonwoori Technology';

	16#00008484:
		F_EtherCAT_VendorIDtoString := 'PHOENIX CONTACT Power Supplies GmbH';

	16#00008562:
		F_EtherCAT_VendorIDtoString := 'Brother Industries Ltd.';

	16#00008632:
		F_EtherCAT_VendorIDtoString := 'Shenzhen Anicetech Automation Company Limited';

	16#00008787:
		F_EtherCAT_VendorIDtoString := 'TESEO spa';

	16#00008800:
		F_EtherCAT_VendorIDtoString := 'Akribis Systems Pte Ltd';

	16#00008818:
		F_EtherCAT_VendorIDtoString := 'Shenyang Machine Tool(Group) Research & Design Institute Co,Ltd. Shanghai Branch';

	16#00008866:
		F_EtherCAT_VendorIDtoString := 'Shanghai DOYEE CNC Technology Co., Ltd.';

	16#00008888:
		F_EtherCAT_VendorIDtoString := 'Changzhou Lead-Motion Intelligent Technology Co., Ltd.';

	16#00008899:
		F_EtherCAT_VendorIDtoString := 'Shandong Laien Optic-Electronic Technology Co., Ltd.';

	16#000088F6:
		F_EtherCAT_VendorIDtoString := 'Harbin Institute of Technology ShenZhen Graduate School';

	16#000088FA:
		F_EtherCAT_VendorIDtoString := 'SIGMATEK GmbH & Co. KG';

	16#00008900:
		F_EtherCAT_VendorIDtoString := 'Genesis Systems, IPG Photonics Company';

	16#00008909:
		F_EtherCAT_VendorIDtoString := 'AIXTRON SE';

	16#00008998:
		F_EtherCAT_VendorIDtoString := 'Shanghai Sumtren Intelligent Technology Co., Ltd.';

	16#00008A8C:
		F_EtherCAT_VendorIDtoString := 'Zhejiang Sci-Tech University, School of Mechanical Engineering and Automation';

	16#00009300:
		F_EtherCAT_VendorIDtoString := 'Shotover Camera Systems LP';

	16#00009320:
		F_EtherCAT_VendorIDtoString := 'Saurer AG, Zweigniederlassung Arbon';

	16#00009403:
		F_EtherCAT_VendorIDtoString := 'Vosch Electronic AG';

	16#00009434:
		F_EtherCAT_VendorIDtoString := 'Shenzhen Hans Motor S&T Co., Ltd.';

	16#00009450:
		F_EtherCAT_VendorIDtoString := 'Zund Systemtechnik AG';

	16#00009496:
		F_EtherCAT_VendorIDtoString := 'Adlos AG';

	16#00009555:
		F_EtherCAT_VendorIDtoString := 'Movensys Inc.';

	16#0000962F:
		F_EtherCAT_VendorIDtoString := 'Sun Fuel Technologies, Inc.';

	16#00009638:
		F_EtherCAT_VendorIDtoString := 'Sungrow Power Supply Co., Ltd.';

	16#000096A9:
		F_EtherCAT_VendorIDtoString := 'Anshi New Energy (Shenzhen) Co., Ltd.';

	16#00009863:
		F_EtherCAT_VendorIDtoString := 'ViE Technologies Sdn. Bhd.';

	16#00009988:
		F_EtherCAT_VendorIDtoString := 'Suzhou Ticbel Direct Drive Motor Co.,Ltd.';

	16#00009999:
		F_EtherCAT_VendorIDtoString := 'Amoy Dynamics (Xiamen) Co., Ltd.';

	16#00009A9A:
		F_EtherCAT_VendorIDtoString := 'Xian Jiaotong University, School of Electronic and Information Engineering';

	16#0000A007:
		F_EtherCAT_VendorIDtoString := 'Shenzhen Hans Scanner S&T Co., Ltd.';

	16#0000A0B6:
		F_EtherCAT_VendorIDtoString := 'Sanritz Automation Co., Ltd.';

	16#0000A0FB:
		F_EtherCAT_VendorIDtoString := 'Toray Engineering D Solutions Co., Ltd.';

	16#0000A1AA:
		F_EtherCAT_VendorIDtoString := 'Shanghai AIM Intelligence Technologies Co., Ltd.';

	16#0000A2A2:
		F_EtherCAT_VendorIDtoString := 'MDSI Ventures LLC';

	16#0000A600:
		F_EtherCAT_VendorIDtoString := 'ASIX s.r.o.';

	16#0000A75E:
		F_EtherCAT_VendorIDtoString := 'ATSE. LLC';

	16#0000A8A8:
		F_EtherCAT_VendorIDtoString := 'Zhejiang CHINT Electrics Co., Ltd.';

	16#0000A8AA:
		F_EtherCAT_VendorIDtoString := 'FUDA Intelligent Systems';

	16#0000AA00:
		F_EtherCAT_VendorIDtoString := 'HATATECH CO., LTD.';

	16#0000AA77:
		F_EtherCAT_VendorIDtoString := 'Muscle Corporation';

	16#0000AAAA:
		F_EtherCAT_VendorIDtoString := 'HIWIN MIKROSYSTEM CORP.';

	16#0000AABB:
		F_EtherCAT_VendorIDtoString := 'GuangZhou Ronsuo Electronic Technology Co.,Ltd';

	16#0000AACC:
		F_EtherCAT_VendorIDtoString := 'Mega-Fabs Motion Systems Ltd. (A Hiwin Company)';

	16#0000AAEC:
		F_EtherCAT_VendorIDtoString := 'AXIMETRIX Automation Inc.';

	16#0000AB57:
		F_EtherCAT_VendorIDtoString := 'RMIT University, School of Electrical and Computer Engineering';

	16#0000ABAB:
		F_EtherCAT_VendorIDtoString := 'Beijing Juntai Tiancheng Technology Co., Ltd.';

	16#0000ABBA:
		F_EtherCAT_VendorIDtoString := 'Triamec Motion AG';

	16#0000ABCD:
		F_EtherCAT_VendorIDtoString := 'SoftEnergy Controls Inc';

	16#0000AC00:
		F_EtherCAT_VendorIDtoString := 'ifm software gmbh';

	16#0000ACC0:
		F_EtherCAT_VendorIDtoString := 'Accutron Ltd';

	16#0000ACDC:
		F_EtherCAT_VendorIDtoString := 'Warp9 Tech Design Inc.';

	16#0000AD84:
		F_EtherCAT_VendorIDtoString := 'Topcon Precision Agriculture';

	16#0000ADDA:
		F_EtherCAT_VendorIDtoString := 'Fraunhofer-Institut fur Lasertechnik (ILT)';

	16#0000ADE5:
		F_EtherCAT_VendorIDtoString := 'ADVES GmbH & Co. KG';

	16#0000AED0:
		F_EtherCAT_VendorIDtoString := 'ANEDO Ltd.';

	16#0000AF1E:
		F_EtherCAT_VendorIDtoString := 'Alpine Racing Ltd';

	16#0000AFEC:
		F_EtherCAT_VendorIDtoString := 'Galaxy Far East Corp.';

	16#0000AFFE:
		F_EtherCAT_VendorIDtoString := 'YASKAWA Europe GmbH';

	16#0000B02A:
		F_EtherCAT_VendorIDtoString := 'Orsys Orth System GmbH';

	16#0000B07A:
		F_EtherCAT_VendorIDtoString := 'Bota Systems AG';

	16#0000B0CE:
		F_EtherCAT_VendorIDtoString := 'Viveris Technologies';

	16#0000B5C2:
		F_EtherCAT_VendorIDtoString := 'Shenzhen Capstone Motion Drive Co., Ltd.';

	16#0000B7A8:
		F_EtherCAT_VendorIDtoString := 'Heinzinger Automotive GmbH';

	16#0000BB80:
		F_EtherCAT_VendorIDtoString := 'Sensa automatisering BV';

	16#0000BBAA:
		F_EtherCAT_VendorIDtoString := 'B. Braun Avitum AG';

	16#0000BBBB:
		F_EtherCAT_VendorIDtoString := 'Sumden Tech Co., Ltd.';

	16#0000BC00:
		F_EtherCAT_VendorIDtoString := 'Brainchild Electronic Co., Ltd.';

	16#0000BD00:
		F_EtherCAT_VendorIDtoString := 'Boston Dynamics, Inc';

	16#0000BE7A:
		F_EtherCAT_VendorIDtoString := 'BETA Dyn GmbH & Co. KG';

	16#0000BEBE:
		F_EtherCAT_VendorIDtoString := 'G.D SpA';

	16#0000BEEF:
		F_EtherCAT_VendorIDtoString := 'National Radio Astronomy Observatory';

	16#0000C00F:
		F_EtherCAT_VendorIDtoString := 'ControlWorks, Inc.';

	16#0000C0DE:
		F_EtherCAT_VendorIDtoString := 'Riedl GmbH';

	16#0000C0FE:
		F_EtherCAT_VendorIDtoString := 'flexlog GmbH';

	16#0000C0FF:
		F_EtherCAT_VendorIDtoString := 'Cohu, Inc.';

	16#0000C15A:
		F_EtherCAT_VendorIDtoString := 'CISA Intelligent Systems & Automation S.L.';

	16#0000C918:
		F_EtherCAT_VendorIDtoString := 'Jiangsu CPTEK Servo Technology Co.Ltd.';

	16#0000CAAA:
		F_EtherCAT_VendorIDtoString := 'Curiosis Inc.';

	16#0000CAFE:
		F_EtherCAT_VendorIDtoString := 'SOTEC Software Entwicklungs GmbH + Co. Mikrocomputertechnik KG';

	16#0000CDCD:
		F_EtherCAT_VendorIDtoString := 'Shenzhen Chengkong Electronics Co., Ltd.';

	16#0000CDEF:
		F_EtherCAT_VendorIDtoString := 'CDEF, Inc.';

	16#0000CEBA:
		F_EtherCAT_VendorIDtoString := 'KEBA Industrial Automation GmbH';

	16#0000D00F:
		F_EtherCAT_VendorIDtoString := 'FRAKO Kondensatoren- und Anlagenbau GmbH';

	16#0000D111:
		F_EtherCAT_VendorIDtoString := 'Wuhan Guide Technology Co., Ltd.';

	16#0000DAB0:
		F_EtherCAT_VendorIDtoString := 'DABO Corporation';

	16#0000DCAC:
		F_EtherCAT_VendorIDtoString := 'Seoul National University, Department of Electrical and Computer Engineering, Power Conversion Systems Laboratory';

	16#0000DE88:
		F_EtherCAT_VendorIDtoString := 'Dalian University of Technology';

	16#0000DEDA:
		F_EtherCAT_VendorIDtoString := 'Potomac Electric Corporation';

	16#0000E0EE:
		F_EtherCAT_VendorIDtoString := 'Marel Hf.';

	16#0000E5AB:
		F_EtherCAT_VendorIDtoString := 'ESAB Welding & Cutting GmbH';

	16#0000EAEA:
		F_EtherCAT_VendorIDtoString := 'meastream GmbH';

	16#0000ECA7:
		F_EtherCAT_VendorIDtoString := 'Emmission';

	16#0000EEEC:
		F_EtherCAT_VendorIDtoString := 'Guangzhou Eichi Technology Co., Ltd.';

	16#0000EEEE:
		F_EtherCAT_VendorIDtoString := 'Willow Garage, Inc.';

	16#0000EF56:
		F_EtherCAT_VendorIDtoString := 'TA Instruments - Waters LLC';

	16#0000EFFE:
		F_EtherCAT_VendorIDtoString := 'Shanghai Passiontech Information Technology Co., Ltd.';

	16#0000F00D:
		F_EtherCAT_VendorIDtoString := 'Hyphen Technologies, Inc.';

	16#0000F0CA:
		F_EtherCAT_VendorIDtoString := 'Imagos S.a.s di Renato Andreola e C.';

	16#0000F1F1:
		F_EtherCAT_VendorIDtoString := 'Red Bull Technology Ltd.';

	16#0000F4F4:
		F_EtherCAT_VendorIDtoString := 'fos4X GmbH';

	16#0000F666:
		F_EtherCAT_VendorIDtoString := 'National Yunlin University of Science and Technology, College of Engineering';

	16#0000F888:
		F_EtherCAT_VendorIDtoString := 'GMT GLOBAL INC.';

	16#0000FAB9:
		F_EtherCAT_VendorIDtoString := 'Fab-9 Corporation';

	16#0000FACE:
		F_EtherCAT_VendorIDtoString := 'Korea Institute of Robot and Convergence (KIRO)';

	16#0000FE09:
		F_EtherCAT_VendorIDtoString := 'Interroll Trommelmotoren GmbH';

	16#0000FEDC:
		F_EtherCAT_VendorIDtoString := 'Silica, Avnet EMG GmbH';

	16#0000FF01:
		F_EtherCAT_VendorIDtoString := 'Innospire Electro Tech Pvt Ltd';

	16#0000FF66:
		F_EtherCAT_VendorIDtoString := 'Harbin Institute of Technology';

	16#0000FFFE:
		F_EtherCAT_VendorIDtoString := 'UENO SEIKI Co.,LTD.';

	16#0000FFAA:
		F_EtherCAT_VendorIDtoString := 'RB3D';

	16#0000FFF1:
		F_EtherCAT_VendorIDtoString := 'BTHL Equipment (Beijing) Co., Ltd.';

	16#0000FFFF:
		F_EtherCAT_VendorIDtoString := 'Robotiq Inc.';

	16#00010000:
		F_EtherCAT_VendorIDtoString := 'Zhejiang Alpha Automotive Technology Co., Ltd.';

	16#00010001:
		F_EtherCAT_VendorIDtoString := 'Hitachi Terminal Mechatronics, Corp.';

	16#00010002:
		F_EtherCAT_VendorIDtoString := 'Dr. Bohrer Lasertec GmbH';

	16#00010100:
		F_EtherCAT_VendorIDtoString := 'Suzhou Jodell Robotics Co., Ltd.';

	16#00010101:
		F_EtherCAT_VendorIDtoString := 'Glidewell Laboratories';

	16#00010123:
		F_EtherCAT_VendorIDtoString := 'AV Electronics S.r.l. a socio unico';

	16#00010150:
		F_EtherCAT_VendorIDtoString := 'MACS World, Inc.';

	16#00010151:
		F_EtherCAT_VendorIDtoString := 'Beijing SaintWise Intelligent Technology Development co.LTD';

	16#00010203:
		F_EtherCAT_VendorIDtoString := 'Jiangsu Kaiserdrive Intelligent Technology Co., Ltd.';

	16#00010205:
		F_EtherCAT_VendorIDtoString := 'Tashang Semiconductor (Shanghai) Co., Ltd.';

	16#0001023E:
		F_EtherCAT_VendorIDtoString := 'Netvision Telecom Inc.';

	16#00010305:
		F_EtherCAT_VendorIDtoString := 'ShenZhen Leadingchips Technology Co.,Ltd';

	16#00010462:
		F_EtherCAT_VendorIDtoString := 'Zhengzhou University of Light Industry, School of Electrical and Information Engineering';

	16#00010502:
		F_EtherCAT_VendorIDtoString := 'Beijing Sunwise Space Technology Co., Ltd.';

	16#00010608:
		F_EtherCAT_VendorIDtoString := 'Shenzhen Jiayu Mechatronic Co., Ltd.';

	16#00010766:
		F_EtherCAT_VendorIDtoString := 'Renesas Electronics (China) Co., Ltd.';

	16#00010780:
		F_EtherCAT_VendorIDtoString := 'Servotecnica SpA';

	16#00010816:
		F_EtherCAT_VendorIDtoString := 'İleri Denetleyici Teknolojiler Mekatronik San. ve Tic. Ltd. Şti.';

	16#00011107:
		F_EtherCAT_VendorIDtoString := 'Utthunga Technologies Pvt. Ltd.';

	16#00011111:
		F_EtherCAT_VendorIDtoString := 'Beijing University of Posts and Telecommunications, School of Automation';

	16#00011211:
		F_EtherCAT_VendorIDtoString := 'BeiJing ETOUCH Technology CO.,LTD.';

	16#000116C7:
		F_EtherCAT_VendorIDtoString := 'Zhejiang Hechuan Technology Co.,Ltd.';

	16#00011975:
		F_EtherCAT_VendorIDtoString := 'Oraklar Yazılım Otomasyon San. ve Tic. Ltd. Şti';

	16#00012550:
		F_EtherCAT_VendorIDtoString := 'KERAjet S.A.';

	16#00012555:
		F_EtherCAT_VendorIDtoString := 'PROAUT TECHNOLOGY GmbH';

	16#00013930:
		F_EtherCAT_VendorIDtoString := 'DANAM SYSTEMS INC.';

	16#000144AB:
		F_EtherCAT_VendorIDtoString := 'Carl Zeiss Optotechnik GmbH';

	16#00015354:
		F_EtherCAT_VendorIDtoString := 'Zhihui Shengda (Beijing) Technology Co., Ltd.';

	16#00015422:
		F_EtherCAT_VendorIDtoString := 'ALPHA MOTION CO., LTD.';

	16#00018843:
		F_EtherCAT_VendorIDtoString := 'M8M Private Limited';

	16#0001DA7A:
		F_EtherCAT_VendorIDtoString := 'MonoDAQ d.o.o.';

	16#0001F001:
		F_EtherCAT_VendorIDtoString := 'EN Technologies Inc.';

	16#00020608:
		F_EtherCAT_VendorIDtoString := 'Harbin Yiao Information Technology Co., Ltd.';

	16#00023155:
		F_EtherCAT_VendorIDtoString := 'Carl Zeiss SMT GmbH';

	16#00028DEC:
		F_EtherCAT_VendorIDtoString := 'Sichuan Dongfang Electric Autocontrol Engineering Co., Ltd.';

	16#00030000:
		F_EtherCAT_VendorIDtoString := 'Dongguan Sindin Precision Instrument Co., Ltd.';

	16#00030004:
		F_EtherCAT_VendorIDtoString := 'XP Power LLC';

	16#00030205:
		F_EtherCAT_VendorIDtoString := 'Levitection Ltd.';

	16#0003030D:
		F_EtherCAT_VendorIDtoString := 'Sioux CCM B.V.';

	16#00030F41:
		F_EtherCAT_VendorIDtoString := 'HUASHENG AUTOMATION CO.,LTD.';

	16#00033332:
		F_EtherCAT_VendorIDtoString := 'Motion Tech Automation, LLC';

	16#00033333:
		F_EtherCAT_VendorIDtoString := 'Amphenol Cable and Interconnect Technologies, Inc.';

	16#00039055:
		F_EtherCAT_VendorIDtoString := 'Sipartek di Marcello Ferri';

	16#00040411:
		F_EtherCAT_VendorIDtoString := 'Narranz Soluciones SL';

	16#00040716:
		F_EtherCAT_VendorIDtoString := 'SYSWORK CO.,LTD.';

	16#00041101:
		F_EtherCAT_VendorIDtoString := 'GuangZhou Xing Hao Precision Technology Company LTD';

	16#00041415:
		F_EtherCAT_VendorIDtoString := 'Harmuth Elektronik GmbH';

	16#00048186:
		F_EtherCAT_VendorIDtoString := 'Intra Corporation';

	16#0004EEE8:
		F_EtherCAT_VendorIDtoString := 'Shanghai ZLAN Information Technology Co., Ltd';

	16#00050903:
		F_EtherCAT_VendorIDtoString := 'Guangdong OPPO Mobile Telecommunications Corp.,Ltd.';

	16#00050D6D:
		F_EtherCAT_VendorIDtoString := 'Rohde & Schwarz GmbH & Co. KG';

	16#00051319:
		F_EtherCAT_VendorIDtoString := 'Generator Research Limited';

	16#000516C2:
		F_EtherCAT_VendorIDtoString := 'Hunan Superstring Technology Co.,Ltd.';

	16#00051C4B:
		F_EtherCAT_VendorIDtoString := 'SICK, Inc.';

	16#00053258:
		F_EtherCAT_VendorIDtoString := 'Shenzhen Encom Electric Technologies Co., Ltd.';

	16#0005AE41:
		F_EtherCAT_VendorIDtoString := 'SAEKI Robotics AG';

	16#00060688:
		F_EtherCAT_VendorIDtoString := 'China Wide Prevention Telecom Technology Co.,Ltd.';

	16#00064541:
		F_EtherCAT_VendorIDtoString := 'R&D Robotics';

	16#00066570:
		F_EtherCAT_VendorIDtoString := 'LG Electronics Inc.';

	16#00069420:
		F_EtherCAT_VendorIDtoString := 'NorthPrint3D';

	16#00070707:
		F_EtherCAT_VendorIDtoString := 'Sodick America Corp.';

	16#00073188:
		F_EtherCAT_VendorIDtoString := 'Hunan Matrix Electronic Technology Co., Ltd.';

	16#00074074:
		F_EtherCAT_VendorIDtoString := 'Roll-2-Roll Technologies LLC';

	16#00074076:
		F_EtherCAT_VendorIDtoString := 'SIC! Software GmbH';

	16#00074855:
		F_EtherCAT_VendorIDtoString := 'LAPPLE AG';

	16#00075500:
		F_EtherCAT_VendorIDtoString := 'ShenZhen Tongchuan Technology Co.,Ltd';

	16#00076761:
		F_EtherCAT_VendorIDtoString := 'ITK Engineering GmbH';

	16#00077054:
		F_EtherCAT_VendorIDtoString := 'EndoQuest Robotics, Inc.';

	16#00077777:
		F_EtherCAT_VendorIDtoString := 'Shanghai Sinyo Electronics Co.,Ltd.';

	16#00080301:
		F_EtherCAT_VendorIDtoString := 'CK Precision Instrument';

	16#00080A0C:
		F_EtherCAT_VendorIDtoString := 'Xian Puyuan Industrial Technology Co., Ltd.';

	16#00080ABC:
		F_EtherCAT_VendorIDtoString := 'Shenzhen XJCSENSOR Technology Co., Ltd.';

	16#00088326:
		F_EtherCAT_VendorIDtoString := 'Willig Embedded Software';

	16#00088888:
		F_EtherCAT_VendorIDtoString := 'Alexan Tech. Inc.';

	16#00090130:
		F_EtherCAT_VendorIDtoString := 'Exvision Corporation';

	16#00090588:
		F_EtherCAT_VendorIDtoString := 'Guangzhou YanWei Electronic Technology Co., Ltd.';

	16#00090606:
		F_EtherCAT_VendorIDtoString := 'Tex Computer SRL';

	16#00090802:
		F_EtherCAT_VendorIDtoString := 'Suzhou EastTech Electronics Co.,Ltd';

	16#00090909:
		F_EtherCAT_VendorIDtoString := 'AONE TECHNOLOGY CO.,LTD.';

	16#00099099:
		F_EtherCAT_VendorIDtoString := 'Nanjing Daqo Electrical Institute Co., Ltd.';

	16#000A000A:
		F_EtherCAT_VendorIDtoString := 'Dongguan Morikawa Motor Technology Co., Ltd.';

	16#000A05E5:
		F_EtherCAT_VendorIDtoString := 'KOSES Co.,Ltd';

	16#000A1016:
		F_EtherCAT_VendorIDtoString := 'Seoul National University of Science and Technology, College of Engineering, Department of Mechanical System and Design Engineering';

	16#000A17AD:
		F_EtherCAT_VendorIDtoString := 'AITAD GmbH';

	16#000A2735:
		F_EtherCAT_VendorIDtoString := 'Shanghai Formal-Tech Information Technology Co., Ltd.';

	16#000A4D7A:
		F_EtherCAT_VendorIDtoString := 'Warsaw University of Technology, Faculty of Electrical Engineering';

	16#000A7B00:
		F_EtherCAT_VendorIDtoString := 'Cornelius Consult';

	16#000AAAAA:
		F_EtherCAT_VendorIDtoString := 'Shandong SIASUN Industrial Software Research Institute Co., Ltd.';

	16#000AAAEC:
		F_EtherCAT_VendorIDtoString := 'AITEC Corporation';

	16#000AB1DE:
		F_EtherCAT_VendorIDtoString := 'The Dude Abides LLC dba Lensrentals.com';

	16#000ABABE:
		F_EtherCAT_VendorIDtoString := 'STECHOQ ROBOTIKA INDONESIA, PT';

	16#000ABCDE:
		F_EtherCAT_VendorIDtoString := 'ASU PRO LLC';

	16#000ACADE:
		F_EtherCAT_VendorIDtoString := 'Istituto Nazionale di Fisica Nucleare, Laboratori Nationale di Frascati';

	16#000ADC05:
		F_EtherCAT_VendorIDtoString := 'adcos GmbH';

	16#000AEA00:
		F_EtherCAT_VendorIDtoString := 'Borda Teknoloji Bilişim A.Ş.';

	16#000B00B0:
		F_EtherCAT_VendorIDtoString := 'Institute of Physics of the Czech Academy of Sciences';

	16#000BBBBB:
		F_EtherCAT_VendorIDtoString := 'FUTURE LIFE TECHNOLOGY CO., LTD.';

	16#000BE11A:
		F_EtherCAT_VendorIDtoString := 'Quality Firmware and Processes Solutions, LLC';

	16#000C0815:
		F_EtherCAT_VendorIDtoString := 'CGX Intelligent Manufacturing (Wuxi) Co., Ltd.';

	16#000C0B07:
		F_EtherCAT_VendorIDtoString := 'Mantis Robotics Inc.';

	16#000C0C0A:
		F_EtherCAT_VendorIDtoString := 'Palmer Design & Manufacturing Ltd Trading as “Palmer Automation”';

	16#000C0C0C:
		F_EtherCAT_VendorIDtoString := 'YES ENERGY srl';

	16#000C1984:
		F_EtherCAT_VendorIDtoString := 'Chroma ATE Inc.';

	16#000D0B0C:
		F_EtherCAT_VendorIDtoString := 'WUHAN DBLC SCIENCE & TECHNOLOGY CO.,LTD.';

	16#000DE1ED:
		F_EtherCAT_VendorIDtoString := 'Delem B.V.';

	16#000E1048:
		F_EtherCAT_VendorIDtoString := 'Toshiba Transport Engineering Inc.';

	16#000EEEEE:
		F_EtherCAT_VendorIDtoString := 'Electroproject B.V.';

	16#000F1016:
		F_EtherCAT_VendorIDtoString := 'OPVengineering GmbH';

	16#000F1024:
		F_EtherCAT_VendorIDtoString := 'enerpowertech Inc.';

	16#00100000:
		F_EtherCAT_VendorIDtoString := 'Shenzhen Inovance Technology Co., Ltd.';

	16#00100006:
		F_EtherCAT_VendorIDtoString := 'Shenzhen Veinar Technology Co., Ltd.';

	16#00100100:
		F_EtherCAT_VendorIDtoString := 'Cyberlogix Ltd';

	16#00100200:
		F_EtherCAT_VendorIDtoString := 'Shenzhen Institute of Advanced Biomedical Robot Co.,Ltd.';

	16#00100DEF:
		F_EtherCAT_VendorIDtoString := 'Rheinmetall Landsysteme GmbH';

	16#00101998:
		F_EtherCAT_VendorIDtoString := 'Fundacao Amazonica de Amparo a Pesquisa e Desenvolvimento Tecnologico Desembargador Paulo dos Anjos';

	16#00102030:
		F_EtherCAT_VendorIDtoString := 'SERWIS CNC Mariusz Mareczko';

	16#00104104:
		F_EtherCAT_VendorIDtoString := 'SBS Science & Technology Co., Ltd.';

	16#00105041:
		F_EtherCAT_VendorIDtoString := 'Inovance Technology Europe GmbH';

	16#00107627:
		F_EtherCAT_VendorIDtoString := 'BYD Company Limited';

	16#00111001:
		F_EtherCAT_VendorIDtoString := 'Windpute (Jiangsu) Intelligent Technology Co., Ltd';

	16#00111111:
		F_EtherCAT_VendorIDtoString := 'Zhejiang Feida Environmental Science & Technology Co., Ltd.';

	16#00111713:
		F_EtherCAT_VendorIDtoString := 'Robotic Systems Integration, Inc.';

	16#00111ACE:
		F_EtherCAT_VendorIDtoString := 'Shenzhen Coastal Fluid Technology Co., Ltd.';

	16#00112233:
		F_EtherCAT_VendorIDtoString := 'YoungTek Electronics Corp.';

	16#00112299:
		F_EtherCAT_VendorIDtoString := 'MELSİS Elektrik Elektronik Yazılım Donanım Ltd. Şti.';

	16#00113322:
		F_EtherCAT_VendorIDtoString := 'SS Innovations China Co., Ltd.';

	16#00116688:
		F_EtherCAT_VendorIDtoString := 'REYA ELECTRIC CO.,LTD.';

	16#0011AB22:
		F_EtherCAT_VendorIDtoString := 'Zhejiang Sanhua Intelligent Controls Co., Ltd';

	16#00120187:
		F_EtherCAT_VendorIDtoString := 'Beijing Institute of Technology, School of Mechatronical Engineering';

	16#00120331:
		F_EtherCAT_VendorIDtoString := 'UBTECH Robotics Corp.';

	16#00123456:
		F_EtherCAT_VendorIDtoString := 'ERAETECH Co., Ltd.';

	16#001234CC:
		F_EtherCAT_VendorIDtoString := 'Compucare India Pvt. Ltd.';

	16#00123ABC:
		F_EtherCAT_VendorIDtoString := 'Microtech Laboratory Inc.';

	16#00124000:
		F_EtherCAT_VendorIDtoString := 'Automatisation JRT Inc.';

	16#00124816:
		F_EtherCAT_VendorIDtoString := 'Easy Etudes et applications systeme SA';

	16#00126815:
		F_EtherCAT_VendorIDtoString := 'EQ GLOBAL Inc.';

	16#00130103:
		F_EtherCAT_VendorIDtoString := 'LOT CES CO., LTD.';

	16#00130268:
		F_EtherCAT_VendorIDtoString := 'Eule Industrial Robotics GmbH & Co. KG';

	16#00130913:
		F_EtherCAT_VendorIDtoString := 'Dongguan Fextend Precision Technology CO.,Ltd';

	16#00132333:
		F_EtherCAT_VendorIDtoString := 'Sudhir Srivastava Innovations Pvt. Ltd.';

	16#00136013:
		F_EtherCAT_VendorIDtoString := 'Beijing RichAuto S&T Co., Ltd';

	16#00141003:
		F_EtherCAT_VendorIDtoString := 'ULVAC AUTOMATION TAIWAN Inc.';

	16#00141198:
		F_EtherCAT_VendorIDtoString := 'Guangdong Gienso Industrial Technology Co., Ltd.';

	16#00141209:
		F_EtherCAT_VendorIDtoString := 'EIKO SOKKI Co. Ltd.';

	16#00143786:
		F_EtherCAT_VendorIDtoString := 'Meril Life Sciences Pvt. Ltd.';

	16#00147852:
		F_EtherCAT_VendorIDtoString := 'Wuxi Lead Intelligent Equipment CO.,LTD.';

	16#00150306:
		F_EtherCAT_VendorIDtoString := 'Shenyang XBANG Technology Co., Ltd.';

	16#00150510:
		F_EtherCAT_VendorIDtoString := 'tecraise GmbH';

	16#00158158:
		F_EtherCAT_VendorIDtoString := 'Hangzhou Advanced Intelligent Manufacturing Systems Co., Ltd.';

	16#0015E65E:
		F_EtherCAT_VendorIDtoString := 'iseg Spezialelektronik GmbH';

	16#00161718:
		F_EtherCAT_VendorIDtoString := 'Guangzhou Start To Sail Industrial Robot Co.,Ltd.';

	16#00166666:
		F_EtherCAT_VendorIDtoString := 'Digitalhorns Network Technology (SuZhou) Co., Ltd';

	16#00168168:
		F_EtherCAT_VendorIDtoString := 'Kronz (Guangzhou) Electronic Co., LTD';

	16#00168888:
		F_EtherCAT_VendorIDtoString := 'WU-YANG Technology Co., Ltd.';

	16#0016F16F:
		F_EtherCAT_VendorIDtoString := 'Fliegl Agrartechnik GmbH';

	16#00170815:
		F_EtherCAT_VendorIDtoString := 'MUHA INC';

	16#00171010:
		F_EtherCAT_VendorIDtoString := 'NIIC (SUZHOU) TECHNOLOGY CO., LTD.';

	16#00171110:
		F_EtherCAT_VendorIDtoString := 'Zhejiang Reagle Sensing Technology Co., Ltd.';

	16#00171207:
		F_EtherCAT_VendorIDtoString := 'Hongxin (Suzhou) Integrated Circuit Co., Ltd.';

	16#00171717:
		F_EtherCAT_VendorIDtoString := 'Tesotronics (trade name BaxEDM)';

	16#00178200:
		F_EtherCAT_VendorIDtoString := 'SmartRay GmbH';

	16#00180116:
		F_EtherCAT_VendorIDtoString := 'Aether, Inc.';

	16#00180201:
		F_EtherCAT_VendorIDtoString := 'KOMOTEK Co., Ltd.';

	16#00180516:
		F_EtherCAT_VendorIDtoString := 'Beijing Holinks Technology Co., Ltd';

	16#00180522:
		F_EtherCAT_VendorIDtoString := 'Shenzhen iManifold Robot Technology Co., Ltd.';

	16#00180613:
		F_EtherCAT_VendorIDtoString := 'Shenzhen Shenzhixin Technology Co., Ltd.';

	16#00181818:
		F_EtherCAT_VendorIDtoString := 'Ningbo Yunsheng Co., Ltd.';

	16#00188888:
		F_EtherCAT_VendorIDtoString := 'Zhejiang Xianda Technology Co., Ltd.';

	16#001897EC:
		F_EtherCAT_VendorIDtoString := 'Loop Technology Ltd';

	16#00190050:
		F_EtherCAT_VendorIDtoString := 'Kayser-Threde GmbH';

	16#00190556:
		F_EtherCAT_VendorIDtoString := 'AXYZ Automation Inc.';

	16#00190683:
		F_EtherCAT_VendorIDtoString := 'Ege Robotics CNC Makine Elektronik Otomasyon Medikal';

	16#00191231:
		F_EtherCAT_VendorIDtoString := 'Haishun Automation Technology (Huizhou) Co., Ltd.';

	16#001918EE:
		F_EtherCAT_VendorIDtoString := 'Tallinn University of Technology (TUT), Faculty of Information Technology';

	16#001919C5:
		F_EtherCAT_VendorIDtoString := 'Carl Cloos Schweisstechnik GmbH';

	16#001919EE:
		F_EtherCAT_VendorIDtoString := 'Tallinn University of Technology (TUT), Faculty of Information Technology';

	16#001970CC:
		F_EtherCAT_VendorIDtoString := 'Ningbo Hirden Industrial Control System Co., Ltd.';

	16#00198452:
		F_EtherCAT_VendorIDtoString := 'NIHON SEIGYO CO.,LTD.';

	16#00200000:
		F_EtherCAT_VendorIDtoString := 'Shenzhen Farwide Electric Co.,Ltd.';

	16#00200402:
		F_EtherCAT_VendorIDtoString := 'Shenzhen Simphoenix Electric Technology Co., Ltd.';

	16#00200804:
		F_EtherCAT_VendorIDtoString := 'Taotech Technology (Qingdao) Co., Ltd.';

	16#00200810:
		F_EtherCAT_VendorIDtoString := 'Jinan Bodor CNC Machine Co.,Ltd.';

	16#00200924:
		F_EtherCAT_VendorIDtoString := 'ARUM DENTISTRY Co., Ltd.';

	16#00201111:
		F_EtherCAT_VendorIDtoString := 'Glass Expansion Pty Ltd';

	16#00201314:
		F_EtherCAT_VendorIDtoString := 'Beijing HollySys Intelligent Technologies Co., Ltd.';

	16#00201318:
		F_EtherCAT_VendorIDtoString := 'Dongguan SMARTWIN Intelligent Equipment Co., Ltd.';

	16#00201605:
		F_EtherCAT_VendorIDtoString := 'Jenex Technologies';

	16#00201811:
		F_EtherCAT_VendorIDtoString := 'Guangzhou ZHIYUAN Electronics Co., Ltd.';

	16#00201812:
		F_EtherCAT_VendorIDtoString := 'FoShan Syckin Intelligent Technology Co., Ltd';

	16#00201813:
		F_EtherCAT_VendorIDtoString := 'SiQin Intelligent Equipment Technology (ShenZhen) Co., Ltd.';

	16#00201911:
		F_EtherCAT_VendorIDtoString := 'Shenzhen Hans Robot Co., Ltd';

	16#00202008:
		F_EtherCAT_VendorIDtoString := 'Suzhou Micro Actuator Technology Co., Ltd.';

	16#00202009:
		F_EtherCAT_VendorIDtoString := 'Tismo Technology Solutions (P) Ltd';

	16#00202103:
		F_EtherCAT_VendorIDtoString := 'Shenzhen Haipengxin Electronics Co., Ltd.';

	16#00202111:
		F_EtherCAT_VendorIDtoString := 'Shanghai Parterny Technology Co., Ltd.';

	16#00202288:
		F_EtherCAT_VendorIDtoString := 'Jiangsu DINGS Intelligent Control Technology Co., Ltd';

	16#00203040:
		F_EtherCAT_VendorIDtoString := 'meerecompany Inc.';

	16#00210811:
		F_EtherCAT_VendorIDtoString := 'Hunan Fugong Power Technology Co., Ltd.';

	16#00211009:
		F_EtherCAT_VendorIDtoString := 'Hangzhou CubeMars Intelligent Technology Co., Ltd.';

	16#00220110:
		F_EtherCAT_VendorIDtoString := 'Research and Production Plant EKRA';

	16#00220805:
		F_EtherCAT_VendorIDtoString := 'Shanghai Mega-Energy Technology Co., Ltd';

	16#00222120:
		F_EtherCAT_VendorIDtoString := 'Shenzhen Canroon Electrical Appliances Co., Ltd';

	16#00223344:
		F_EtherCAT_VendorIDtoString := 'FPT Software Ltd.';

	16#00224466:
		F_EtherCAT_VendorIDtoString := 'Shenzhen Sinexcel Electric Co., Ltd.';

	16#00228100:
		F_EtherCAT_VendorIDtoString := 'eMotion Co., Ltd.';

	16#00230315:
		F_EtherCAT_VendorIDtoString := 'Proxception GmbH';

	16#00230803:
		F_EtherCAT_VendorIDtoString := 'Shenzhen Yuanhui Intelligent Technology Co., Ltd.';

	16#00231212:
		F_EtherCAT_VendorIDtoString := 'Chongqing Kekai Qianwei Electric Co., Ltd.';

	16#00231523:
		F_EtherCAT_VendorIDtoString := 'KOLTEST Elektronik San. ve Tic. LTD Şti.';

	16#00231970:
		F_EtherCAT_VendorIDtoString := 'HRK-BRK SRLS';

	16#0023EFAB:
		F_EtherCAT_VendorIDtoString := 'Shenzhen ROBOTMETA Technology Co., Ltd.';

	16#00242628:
		F_EtherCAT_VendorIDtoString := 'GuangZhou CHANGEN Electronic Technology Co.,Ltd.';

	16#00250001:
		F_EtherCAT_VendorIDtoString := 'Nanjing Chenguang Group Co., Ltd.';

	16#00250002:
		F_EtherCAT_VendorIDtoString := 'Jiangsu Jinling Institute of Intelligent Manufacturing Co.,Ltd.';

	16#00250993:
		F_EtherCAT_VendorIDtoString := 'Manner Sensortelemetrie GmbH';

	16#00251201:
		F_EtherCAT_VendorIDtoString := 'Hano Manufacturing Co., Ltd.';

	16#00252525:
		F_EtherCAT_VendorIDtoString := 'EODIGITEK Co.,Ltd';

	16#00255210:
		F_EtherCAT_VendorIDtoString := 'SMART TESTSOLUTIONS GmbH';

	16#00260954:
		F_EtherCAT_VendorIDtoString := 'Meinhard Koppitz, Elektronikentwicklung';

	16#00270697:
		F_EtherCAT_VendorIDtoString := 'Alinghi Red Bull Racing Spain SLU';

	16#00270919:
		F_EtherCAT_VendorIDtoString := 'GUREN Design & Engineering';

	16#00289117:
		F_EtherCAT_VendorIDtoString := 'SHENZHEN JINGFENG MEDICAL TECHNOLOGY CO., LTD.';

	16#00290968:
		F_EtherCAT_VendorIDtoString := 'RUAG Defence Deutschland GmbH';

	16#00300077:
		F_EtherCAT_VendorIDtoString := 'Nations Technologies Inc.';

	16#00300354:
		F_EtherCAT_VendorIDtoString := 'Jiangsu Donghua Testing Technology Co., Ltd.';

	16#00308012:
		F_EtherCAT_VendorIDtoString := 'Creasoft SL';

	16#0030AE7B:
		F_EtherCAT_VendorIDtoString := 'Zhejiang Dusun Electron Co., Ltd.';

	16#0030DB07:
		F_EtherCAT_VendorIDtoString := 'Modbot, Inc.';

	16#00310713:
		F_EtherCAT_VendorIDtoString := 'Sruhad Technologies Pvt Ltd';

	16#003111C0:
		F_EtherCAT_VendorIDtoString := 'RJG Inc.';

	16#00314000:
		F_EtherCAT_VendorIDtoString := 'Balance Systems S.r.l.';

	16#00314159:
		F_EtherCAT_VendorIDtoString := 'Weka Robotics Limited';

	16#0031636F:
		F_EtherCAT_VendorIDtoString := 'T1 Co., LTD.';

	16#00323232:
		F_EtherCAT_VendorIDtoString := 'STMicroelectronics International NV';

	16#00330033:
		F_EtherCAT_VendorIDtoString := 'DFI Inc.';

	16#00333999:
		F_EtherCAT_VendorIDtoString := 'AirSack (Wuxi) Electronic Technology Co., Ltd.';

	16#00334658:
		F_EtherCAT_VendorIDtoString := 'CaTs3 Limited';

	16#00335160:
		F_EtherCAT_VendorIDtoString := 'Precision Technology Corporation';

	16#00335233:
		F_EtherCAT_VendorIDtoString := 'Shanghai HOCH Laser Technology Co., Ltd.';

	16#00340702:
		F_EtherCAT_VendorIDtoString := 'Shanghai Rui Fast Automation Equipment Co.,Ltd.';

	16#00345588:
		F_EtherCAT_VendorIDtoString := 'UTECHZONE CO., LTD.';

	16#00345678:
		F_EtherCAT_VendorIDtoString := 'ABB Beijing Drive Systems Co., Ltd.';

	16#00345869:
		F_EtherCAT_VendorIDtoString := 'APE Technology Co., Ltd.';

	16#00351090:
		F_EtherCAT_VendorIDtoString := 'Zhejiang Dafeng Industry Co., Ltd.';

	16#00361300:
		F_EtherCAT_VendorIDtoString := 'Egle Systems S.L.';

	16#00369369:
		F_EtherCAT_VendorIDtoString := 'Honeywell Technology Solutions Lab Private Limited';

	16#0039544C:
		F_EtherCAT_VendorIDtoString := '9T Labs AG';

	16#003C6F3A:
		F_EtherCAT_VendorIDtoString := 'NeoHealthTechnology, LTD.';

	16#00400000:
		F_EtherCAT_VendorIDtoString := 'Suzhou Anchi Control System Co., Ltd.';

	16#00404040:
		F_EtherCAT_VendorIDtoString := 'ViewMove Technologies Inc.';

	16#004083A9:
		F_EtherCAT_VendorIDtoString := 'Deutsches Elektronen-Synchrotron DESY';

	16#00410041:
		F_EtherCAT_VendorIDtoString := 'Ayoff Industrial Technologies Inc.';

	16#00410222:
		F_EtherCAT_VendorIDtoString := 'Changzhou Jinzhi Drive Technology Co., Ltd.';

	16#0041334D:
		F_EtherCAT_VendorIDtoString := 'A3M-Ingenieurgesellschaft mbH';

	16#00414141:
		F_EtherCAT_VendorIDtoString := 'Bruker Technologies Ltd.';

	16#00414243:
		F_EtherCAT_VendorIDtoString := 'Jiangxi Anbaichuan Electric Co., Ltd.';

	16#0041444C:
		F_EtherCAT_VendorIDtoString := 'ADL Analoge und Digitale Leistungselektronik GmbH';

	16#0041444D:
		F_EtherCAT_VendorIDtoString := 'Adullam Tech Co., Ltd.';

	16#00414458:
		F_EtherCAT_VendorIDtoString := 'ADX Systems SA';

	16#00414853:
		F_EtherCAT_VendorIDtoString := 'Riole Eletronica Ltda';

	16#00414953:
		F_EtherCAT_VendorIDtoString := 'AI Solutions 87 LLC';

	16#00414C54:
		F_EtherCAT_VendorIDtoString := 'ALTIMA Corp.';

	16#00414E59:
		F_EtherCAT_VendorIDtoString := 'ANYbotics AG';

	16#00415041:
		F_EtherCAT_VendorIDtoString := 'APA Sp. z o.o.';

	16#00415049:
		F_EtherCAT_VendorIDtoString := 'Teledyne API';

	16#0041504C:
		F_EtherCAT_VendorIDtoString := 'APL Automobil-Pruftechnik Landau GmbH';

	16#00415450:
		F_EtherCAT_VendorIDtoString := 'Atonarp Inc.';

	16#00416C78:
		F_EtherCAT_VendorIDtoString := 'AiLux S.r.l.';

	16#00418108:
		F_EtherCAT_VendorIDtoString := 'Shanghai Xiangshi Intelligent Technology Co.,Ltd.';

	16#00424242:
		F_EtherCAT_VendorIDtoString := 'European X-Ray Free-Electron Laser Facility GmbH';

	16#00424345:
		F_EtherCAT_VendorIDtoString := 'Seren Industrial Power Systems, Inc.';

	16#00424D54:
		F_EtherCAT_VendorIDtoString := 'Burghart Messtechnik GmbH';

	16#00425343:
		F_EtherCAT_VendorIDtoString := 'L3 Commercial Training Solutions (Aerosim Technologies, INC)';

	16#00434954:
		F_EtherCAT_VendorIDtoString := 'Chiba Institute of Technology (CIT)';

	16#00434D45:
		F_EtherCAT_VendorIDtoString := 'Cambridge Micro Engineering Limited';

	16#00434D4E:
		F_EtherCAT_VendorIDtoString := 'CIMON CO.,LTD.';

	16#00435452:
		F_EtherCAT_VendorIDtoString := 'Controlar - Electronica Industrial e Sistemas, S.A.';

	16#00442656:
		F_EtherCAT_VendorIDtoString := 'D&V Electronics Ltd.';

	16#00444444:
		F_EtherCAT_VendorIDtoString := 'Eltech Ltd.';

	16#00444543:
		F_EtherCAT_VendorIDtoString := 'Nanjing DECOWELL Automation Co., Ltd';

	16#00444949:
		F_EtherCAT_VendorIDtoString := 'DISTek Integration, Inc.';

	16#00444950:
		F_EtherCAT_VendorIDtoString := 'Astrodyne TDI';

	16#00444D53:
		F_EtherCAT_VendorIDtoString := 'Suzhou DHMS Information Technology Co.,Ltd.';

	16#00444D54:
		F_EtherCAT_VendorIDtoString := 'Dematic Corp.';

	16#00445341:
		F_EtherCAT_VendorIDtoString := 'DS AUTOMOTION GmbH';

	16#00445345:
		F_EtherCAT_VendorIDtoString := 'Daewoo Shipbuilding & Marine Engineering Co., Ltd.';

	16#00445653:
		F_EtherCAT_VendorIDtoString := 'Shenzhen DVS Mechatronics Co., Ltd.';

	16#00448976:
		F_EtherCAT_VendorIDtoString := 'Busch Manufacturing Korea, Ltd.';

	16#00454854:
		F_EtherCAT_VendorIDtoString := 'Eagle Harbor Technologies Inc.';

	16#00455341:
		F_EtherCAT_VendorIDtoString := 'Embedded Systems Academy, Inc.';

	16#00455354:
		F_EtherCAT_VendorIDtoString := 'Steinbeis Embedded Systems Technologies GmbH';

	16#00455443:
		F_EtherCAT_VendorIDtoString := 'Electronic Theatre Controls, Inc.';

	16#00455453:
		F_EtherCAT_VendorIDtoString := 'ITMO University, Department of Control Systems and Industrial Robotics, Chair of Electrical Engineering and Precision Electromechanical Systems';

	16#0045564F:
		F_EtherCAT_VendorIDtoString := 'Evolution Measurement Ltd.';

	16#00455A43:
		F_EtherCAT_VendorIDtoString := 'Shandong EZCode Intelligent Technology Co., Ltd.';

	16#00456789:
		F_EtherCAT_VendorIDtoString := 'SKY TECHNOLOGY DEVELOPMENT CO.,LTD. CHINESE ACADEMY OF SCIENCES';

	16#00456E76:
		F_EtherCAT_VendorIDtoString := 'Envision Energy (Jiangsu) CO., LTD.';

	16#00462650:
		F_EtherCAT_VendorIDtoString := 'F&P Robotics AG';

	16#00465554:
		F_EtherCAT_VendorIDtoString := 'Future Electronics Inc.';

	16#004711BB:
		F_EtherCAT_VendorIDtoString := 'Moehwald GmbH';

	16#00474253:
		F_EtherCAT_VendorIDtoString := 'GBS Elektronik GmbH';

	16#0047494E:
		F_EtherCAT_VendorIDtoString := 'Ginolis Oy';

	16#00474E44:
		F_EtherCAT_VendorIDtoString := 'Shanghai GND eTech Co., Ltd.';

	16#00475349:
		F_EtherCAT_VendorIDtoString := 'GSI GeoSolutions International Ltd';

	16#00475354:
		F_EtherCAT_VendorIDtoString := 'Global Standard Technology Co., Ltd.';

	16#00475435:
		F_EtherCAT_VendorIDtoString := 'Gate5 GmbH';

	16#00481417:
		F_EtherCAT_VendorIDtoString := 'Innodelec Sarl';

	16#0048414D:
		F_EtherCAT_VendorIDtoString := 'Hamilton Bonaduz AG';

	16#0048414F:
		F_EtherCAT_VendorIDtoString := 'Shanghai Kepler Exploration Robot Co., Ltd.';

	16#00484D30:
		F_EtherCAT_VendorIDtoString := 'Hexagon Metrology S.p.A.';

	16#0048504D:
		F_EtherCAT_VendorIDtoString := 'HPMicro Semiconductor Co., Ltd.';

	16#00485088:
		F_EtherCAT_VendorIDtoString := 'Shanghai Shenke Technology Co., Ltd.';

	16#00485247:
		F_EtherCAT_VendorIDtoString := 'Neura Robotics GmbH';

	16#00485349:
		F_EtherCAT_VendorIDtoString := 'Headspring Inc.';

	16#0048554B:
		F_EtherCAT_VendorIDtoString := 'Kendrion Kuhnke Automation GmbH';

	16#00485645:
		F_EtherCAT_VendorIDtoString := 'High Voltage Engineering Europa B.V.';

	16#00485653:
		F_EtherCAT_VendorIDtoString := 'HV Sistemas S.L.';

	16#00485749:
		F_EtherCAT_VendorIDtoString := 'Halleck-Willard Incorporated';

	16#00490628:
		F_EtherCAT_VendorIDtoString := 'KYOWA ELECTRONIC INSTRUMENTS  CO., LTD.';

	16#00491617:
		F_EtherCAT_VendorIDtoString := 'FST Co., Ltd.';

	16#00494252:
		F_EtherCAT_VendorIDtoString := 'IBR Messtechnik GmbH & Co. KG';

	16#00494253:
		F_EtherCAT_VendorIDtoString := 'IBS Precision Engineering BV';

	16#00494256:
		F_EtherCAT_VendorIDtoString := 'IBV - Echtzeit- und Embedded GmbH & Co. KG';

	16#00494350:
		F_EtherCAT_VendorIDtoString := 'ICP DAS Co.,Ltd.';

	16#00494458:
		F_EtherCAT_VendorIDtoString := 'IDX Co. Ltd.';

	16#00495253:
		F_EtherCAT_VendorIDtoString := 'IRS Systementwicklung GmbH';

	16#00495254:
		F_EtherCAT_VendorIDtoString := 'IRT SA';

	16#00499816:
		F_EtherCAT_VendorIDtoString := 'Seoul Precision Machines Co., Ltd.';

	16#004A4154:
		F_EtherCAT_VendorIDtoString := 'Jenaer Antriebstechnik GmbH';

	16#004A542E:
		F_EtherCAT_VendorIDtoString := 'JT Corp.';

	16#004A5434:
		F_EtherCAT_VendorIDtoString := 'JT4, LLC';

	16#004B4544:
		F_EtherCAT_VendorIDtoString := 'Kinetic Engineering Design Ltd';

	16#004B4657:
		F_EtherCAT_VendorIDtoString := 'Hangzhou ConfirmWare Technology Co., Ltd.';

	16#004B465A:
		F_EtherCAT_VendorIDtoString := 'Deutsches Krebsforschungszentrum (DKFZ)';

	16#004B4743:
		F_EtherCAT_VendorIDtoString := 'Keisokugiken Corporation';

	16#004B494D:
		F_EtherCAT_VendorIDtoString := 'PRESYS Co., Ltd.';

	16#004B5243:
		F_EtherCAT_VendorIDtoString := 'KAWADA ROBOTICS CORPORATION';

	16#004B525A:
		F_EtherCAT_VendorIDtoString := 'Kriszon Enterprise';

	16#004B6561:
		F_EtherCAT_VendorIDtoString := 'RobCo GmbH';

	16#004C434D:
		F_EtherCAT_VendorIDtoString := 'Linz Center of Mechatronics GmbH';

	16#004C4553:
		F_EtherCAT_VendorIDtoString := 'Lucas Electronic Solutions Pty Ltd';

	16#004C4F43:
		F_EtherCAT_VendorIDtoString := 'KELO Robotics GmbH';

	16#004C545A:
		F_EtherCAT_VendorIDtoString := 'Lithoz GmbH';

	16#004C5552:
		F_EtherCAT_VendorIDtoString := 'University of Oviedo, Electrical, Electronic, Computer and Systems Engineering Department';

	16#004D4153:
		F_EtherCAT_VendorIDtoString := 'AGEMA Germany GmbH';

	16#004D4159:
		F_EtherCAT_VendorIDtoString := 'Chr. Mayr GmbH + Co. KG';

	16#004d4448:
		F_EtherCAT_VendorIDtoString := 'Heidelberger Druckmaschinen AG';

	16#004D4543:
		F_EtherCAT_VendorIDtoString := 'Mecalc PTY Limited';

	16#004D4544:
		F_EtherCAT_VendorIDtoString := 'Meditrina Inc.';

	16#004D4945:
		F_EtherCAT_VendorIDtoString := 'SuperVac Maschinenbau GmbH';

	16#004D5249:
		F_EtherCAT_VendorIDtoString := 'Volga State University of Technology, Faculty of Information Technologies and Computer Engineering';

	16#004D544E:
		F_EtherCAT_VendorIDtoString := 'MOTEON GmbH';

	16#004E4154:
		F_EtherCAT_VendorIDtoString := 'NARAE NANOTECH Corporation';

	16#004E4355:
		F_EtherCAT_VendorIDtoString := 'Nicolaus Copernicus University in Torun (NCU), Faculty of Physics, Astronomy and Informatics';

	16#004E454D:
		F_EtherCAT_VendorIDtoString := 'NEMONOS GmbH';

	16#004E4554:
		F_EtherCAT_VendorIDtoString := 'Wuxi Yikesen Intelligent Technology Co., Ltd.';

	16#004E5044:
		F_EtherCAT_VendorIDtoString := 'North Point Defense, Inc.';

	16#004E5854:
		F_EtherCAT_VendorIDtoString := 'NEXTY Electronics Corporation';

	16#004F4E53:
		F_EtherCAT_VendorIDtoString := 'ONSYS Co., Ltd';

	16#004F5053:
		F_EtherCAT_VendorIDtoString := 'Opsens Inc.';

	16#004F524D:
		F_EtherCAT_VendorIDtoString := 'ORMEC Systems Corp.';

	16#00502654:
		F_EtherCAT_VendorIDtoString := 'POSCO ENGINEERING Co., Ltd.';

	16#00504155:
		F_EtherCAT_VendorIDtoString := 'ONA Electroerosion S.A.';

	16#0050434B:
		F_EtherCAT_VendorIDtoString := 'PC Krause and Associates, Inc.';

	16#0050495A:
		F_EtherCAT_VendorIDtoString := 'Pizzato Elettrica S.r.l.';

	16#00504C45:
		F_EtherCAT_VendorIDtoString := 'Pleora Technologies Inc.';

	16#00504D43:
		F_EtherCAT_VendorIDtoString := 'Ningbo Physis Technology Co.,Ltd.';

	16#0050524F:
		F_EtherCAT_VendorIDtoString := 'PROTEC Co.,Ltd.';

	16#00505344:
		F_EtherCAT_VendorIDtoString := 'Panasonic System Design Co., Ltd.';

	16#00505347:
		F_EtherCAT_VendorIDtoString := 'PowerSparks GmbH';

	16#00505349:
		F_EtherCAT_VendorIDtoString := 'Paul Scherrer Institut';

	16#0050535A:
		F_EtherCAT_VendorIDtoString := 'Packsize Technologies AB';

	16#00505450:
		F_EtherCAT_VendorIDtoString := 'PT Photonic Tools GmbH';

	16#00508280:
		F_EtherCAT_VendorIDtoString := 'SOMA GmbH';

	16#00509188:
		F_EtherCAT_VendorIDtoString := 'Ching Hung Machinery & Electric Industrial Co., Ltd.';

	16#005107EC:
		F_EtherCAT_VendorIDtoString := '5Io.Tech GmbH';

	16#00511018:
		F_EtherCAT_VendorIDtoString := 'NIHON PISCO CO., LTD.';

	16#00515151:
		F_EtherCAT_VendorIDtoString := 'Shanghai VolBoff Electron Science & Technology Co., Ltd.';

	16#00515958:
		F_EtherCAT_VendorIDtoString := 'Shenzhen QianYanXin Electronic Technology Co., Ltd';

	16#00517517:
		F_EtherCAT_VendorIDtoString := 'Shanghai Metro Electronic Technology Co., Ltd.';

	16#00518000:
		F_EtherCAT_VendorIDtoString := 'Fortior Technology (Shenzhen) Co.,Ltd.';

	16#00518888:
		F_EtherCAT_VendorIDtoString := 'Shanghai Rock Technology Co., Ltd.';

	16#00522227:
		F_EtherCAT_VendorIDtoString := 'Titanium Tiger Robot Technology (Shanghai) Co., Ltd.';

	16#00522543:
		F_EtherCAT_VendorIDtoString := 'Shanghai JiQi Robot Technology Co., Ltd.';

	16#00524159:
		F_EtherCAT_VendorIDtoString := 'RAYLASE GmbH';

	16#00524254:
		F_EtherCAT_VendorIDtoString := 'Daegu Gyeongbuk Institute of Science & Technology, Robotics System Research Division';

	16#0052454E:
		F_EtherCAT_VendorIDtoString := 'Renishaw plc';

	16#00524D54:
		F_EtherCAT_VendorIDtoString := 'Rheonik Messtechnik GmbH';

	16#00525349:
		F_EtherCAT_VendorIDtoString := 'Technische Universitat Munchen, Munich Institute of Robotics and Machine Intelligence (MIRMI)';

	16#00528785:
		F_EtherCAT_VendorIDtoString := 'Suzhou Lingchen Acquisition Computer Co., Ltd.';

	16#00532579:
		F_EtherCAT_VendorIDtoString := 'NANORAY Co., Ltd.';

	16#00534147:
		F_EtherCAT_VendorIDtoString := 'Siemens Aktiengesellschaft';

	16#00534543:
		F_EtherCAT_VendorIDtoString := 'Samsung Electronics Co. Ltd.';

	16#00534549:
		F_EtherCAT_VendorIDtoString := 'Sumitomo Electric Industries, Ltd.';

	16#00534649:
		F_EtherCAT_VendorIDtoString := 'Starfire Industries, LLC';

	16#00534652:
		F_EtherCAT_VendorIDtoString := 'SFERA S.r.l.';

	16#00534743:
		F_EtherCAT_VendorIDtoString := 'Skyloom Global Corp.';

	16#00534745:
		F_EtherCAT_VendorIDtoString := 'SG Electronic Systems SRLS';

	16#00534754:
		F_EtherCAT_VendorIDtoString := 'Seiki Global Technology Pte Ltd';

	16#00534A57:
		F_EtherCAT_VendorIDtoString := 'Wuxi Holyview Microelectronics Co., LTD';

	16#00534C4E:
		F_EtherCAT_VendorIDtoString := 'SLN Technologies Pvt. Ltd.';

	16#00534D45:
		F_EtherCAT_VendorIDtoString := 'SimpleMotion Pty Ltd';

	16#00534E4E:
		F_EtherCAT_VendorIDtoString := 'Smith & Nephew, Inc.';

	16#00534E50:
		F_EtherCAT_VendorIDtoString := 'Marmatek Muhendislik Endustriyel Test Olcum ve Otomasyon San. ve Tic. Ltd. Sti.';

	16#00534F4D:
		F_EtherCAT_VendorIDtoString := 'SOMIC Verpackungsmaschinen GmbH & Co. KG';

	16#00535044:
		F_EtherCAT_VendorIDtoString := 'Simplexity Product Development, Inc.';

	16#00535349:
		F_EtherCAT_VendorIDtoString := 'SSI CO.,LTD.';

	16#00535445:
		F_EtherCAT_VendorIDtoString := 'SMITEC S.p.A.';

	16#0053554E:
		F_EtherCAT_VendorIDtoString := 'SUNSAY GENERIC CO., LTD.';

	16#00536D61:
		F_EtherCAT_VendorIDtoString := 'SmarAct GmbH';

	16#00544543:
		F_EtherCAT_VendorIDtoString := 'TECHMETA ENGINEERING SAS';

	16#00544544:
		F_EtherCAT_VendorIDtoString := 'Tokyo Electron Kyushu Limited';

	16#0054454B:
		F_EtherCAT_VendorIDtoString := 'Toray Engineering Co., Ltd.';

	16#0054454C:
		F_EtherCAT_VendorIDtoString := 'Tokyo Electron Limited';

	16#0054454D:
		F_EtherCAT_VendorIDtoString := 'Tem-Tech Lab.';

	16#00544855:
		F_EtherCAT_VendorIDtoString := 'Technische Hochschule Ulm, Fakultat fur Mechatronik und Medizintechnik';

	16#00544D45:
		F_EtherCAT_VendorIDtoString := 'TOMEN ELECTRONICS CORPORATION';

	16#00544E47:
		F_EtherCAT_VendorIDtoString := 'Technolution B.V.';

	16#00544E4D:
		F_EtherCAT_VendorIDtoString := 'STE Trekwerk B.V.';

	16#00544E5A:
		F_EtherCAT_VendorIDtoString := 'Team New Zealand Limited (Trading as Emirates Team New Zealand)';

	16#00545145:
		F_EtherCAT_VendorIDtoString := 'TRONTEQ Electronic GbR';

	16#00545249:
		F_EtherCAT_VendorIDtoString := 'Techman Robot Inc.';

	16#0054534E:
		F_EtherCAT_VendorIDtoString := 'Suzhou TSN Technology Co., Ltd.';

	16#00545454:
		F_EtherCAT_VendorIDtoString := 'Sakarya University, Faculty of Computer and Information Sciences, Computer Engineering Department';

	16#00546936:
		F_EtherCAT_VendorIDtoString := 'JS Automation Corp.';

	16#00553230:
		F_EtherCAT_VendorIDtoString := 'HD Hyundai Electric Co., Ltd.';

	16#00554549:
		F_EtherCAT_VendorIDtoString := 'United Electronic Industries, Inc.';

	16#0055494D:
		F_EtherCAT_VendorIDtoString := 'United Intelligence Robotics (Zhejiang) Co.,Ltd.';

	16#00554952:
		F_EtherCAT_VendorIDtoString := 'Shanghai United Intelligence Robotics Inc.';

	16#00554C54:
		F_EtherCAT_VendorIDtoString := 'Ultimaker B.V.';

	16#00555555:
		F_EtherCAT_VendorIDtoString := 'Jiangxi Fashion Technology Co., Ltd.';

	16#0055555A:
		F_EtherCAT_VendorIDtoString := 'Korea Institute of Machinery & Materials, Advanced Manufacturing Systems Research Division';

	16#0055555B:
		F_EtherCAT_VendorIDtoString := 'Korea Institute of Machinery & Materials, Nano-Convergence Manufacturing Systems Research Division, Department of Printed Electronics';

	16#00555888:
		F_EtherCAT_VendorIDtoString := 'Zhejiang Shuanghuan Driveline Co., Ltd.';

	16#00555AAA:
		F_EtherCAT_VendorIDtoString := 'Normatech Engineering AG';

	16#00556666:
		F_EtherCAT_VendorIDtoString := 'ShenZhen V&T Technologies Co., Ltd.';

	16#0055AA88:
		F_EtherCAT_VendorIDtoString := 'Dongguan Strong Intelligent Equipment Co., LTD';

	16#00564343:
		F_EtherCAT_VendorIDtoString := 'Volvo Car Group';

	16#00564D49:
		F_EtherCAT_VendorIDtoString := 'VMI Holland B.V.';

	16#00564E54:
		F_EtherCAT_VendorIDtoString := 'Vention Inc.';

	16#00565203:
		F_EtherCAT_VendorIDtoString := 'Shenzhen DOHHO Electric Co., Ltd.';

	16#00568568:
		F_EtherCAT_VendorIDtoString := 'Karma Technology Ltd.';

	16#00574154:
		F_EtherCAT_VendorIDtoString := 'watttron GmbH';

	16#00574654:
		F_EtherCAT_VendorIDtoString := 'Weatherford Oil Tool GmbH';

	16#00574954:
		F_EtherCAT_VendorIDtoString := 'Witium Co., Ltd.';

	16#00577800:
		F_EtherCAT_VendorIDtoString := 'Inca Digital Printers Limited';

	16#00578485:
		F_EtherCAT_VendorIDtoString := 'Cerebrus Corporation';

	16#00584D4D:
		F_EtherCAT_VendorIDtoString := 'Xiamen Micromatch Electronic Information Technology Co.,Ltd.';

	16#005860AE:
		F_EtherCAT_VendorIDtoString := 'Shenzhen Daxinda Mechanical and Electrical Equipment Co., Ltd.';

	16#00587675:
		F_EtherCAT_VendorIDtoString := 'SICHUAN ETROL TECHNOLOGIES CO., LTD.';

	16#00594188:
		F_EtherCAT_VendorIDtoString := 'Shenzhen TianAn Sensor Technology Co.,Ltd';

	16#005A5A5A:
		F_EtherCAT_VendorIDtoString := 'Hangzhou Zhenzheng Robot Technology Co.,LTD';

	16#005A7967:
		F_EtherCAT_VendorIDtoString := 'Zygo Corporation';

	16#005E5E5E:
		F_EtherCAT_VendorIDtoString := 'Ser.mac srl';

	16#005EA71E:
		F_EtherCAT_VendorIDtoString := 'Tethers Unlimited, Inc.';

	16#00600613:
		F_EtherCAT_VendorIDtoString := 'Google LLC';

	16#00600885:
		F_EtherCAT_VendorIDtoString := 'Xiamen Hongfa Electroacoustic Co.,Ltd.';

	16#00616263:
		F_EtherCAT_VendorIDtoString := 'Hangzhou EZVIZ Network Co.,Ltd.';

	16#00616978:
		F_EtherCAT_VendorIDtoString := 'aixcon PowerSystems GmbH';

	16#00616C6C:
		F_EtherCAT_VendorIDtoString := 'Allestec Corporation';

	16#00618618:
		F_EtherCAT_VendorIDtoString := 'Panasonic Software Development Center Dalian Co., Ltd.';

	16#00618913:
		F_EtherCAT_VendorIDtoString := 'TECHEST Co.,Ltd.';

	16#00620278:
		F_EtherCAT_VendorIDtoString := 'APHA AUTOMATE CO., LTD.';

	16#0062696F:
		F_EtherCAT_VendorIDtoString := 'Harmonic Bionics, Inc.';

	16#0062AE2D:
		F_EtherCAT_VendorIDtoString := 'Redstone Aerospace Corporation';

	16#0063756D:
		F_EtherCAT_VendorIDtoString := 'Imagen Energy Inc.';

	16#00640627:
		F_EtherCAT_VendorIDtoString := 'MORNSUN Guangzhou Science & Technology Co., Ltd.';

	16#00643000:
		F_EtherCAT_VendorIDtoString := 'Maple Electronics';

	16#00654321:
		F_EtherCAT_VendorIDtoString := 'YUCHANG TECH Co., Ltd.';

	16#0065726F:
		F_EtherCAT_VendorIDtoString := 'ZeroErr Control Co.,Ltd';

	16#00660066:
		F_EtherCAT_VendorIDtoString := 'Ningbo Zhafir Plastics Machinery Co., LTD.';

	16#00660088:
		F_EtherCAT_VendorIDtoString := 'Ningbo Haitian Precision Machinery Co., Ltd.';

	16#00661100:
		F_EtherCAT_VendorIDtoString := 'Shanghai JAKA Robotics Ltd.';

	16#00666666:
		F_EtherCAT_VendorIDtoString := 'Changzhou MVision IT Technology Co., Ltd.';

	16#00666888:
		F_EtherCAT_VendorIDtoString := 'Hunan Sharing Intelligent Machines Co., Ltd.';

	16#00666999:
		F_EtherCAT_VendorIDtoString := 'Shenzhen Motion G Intelligent Technology Co., Ltd.';

	16#00667675:
		F_EtherCAT_VendorIDtoString := 'Bilko Computer Control & Automation Co.';

	16#00667788:
		F_EtherCAT_VendorIDtoString := 'Zhejiang Nseptstars Technology Co., Ltd.';

	16#00668899:
		F_EtherCAT_VendorIDtoString := 'Nanjing Hi-Speedlink Technology Co., Ltd.';

	16#00669988:
		F_EtherCAT_VendorIDtoString := 'Wuhan NEWLAS Intelligent Technology Co., Ltd.';

	16#00678382:
		F_EtherCAT_VendorIDtoString := 'Cornerstone Robotics Limited';

	16#00678384:
		F_EtherCAT_VendorIDtoString := 'Cornerstone Technology (Shenzhen) Limited';

	16#00681168:
		F_EtherCAT_VendorIDtoString := 'Kinco Electric (Shenzhen) Ltd.';

	16#00685051:
		F_EtherCAT_VendorIDtoString := 'INTERACT Inc.';

	16#00686868:
		F_EtherCAT_VendorIDtoString := 'Chengdu GUNT Weida CNC Technology Co., Ltd.';

	16#00688165:
		F_EtherCAT_VendorIDtoString := 'EFORT Intelligent Equipment Co., Ltd.';

	16#00688191:
		F_EtherCAT_VendorIDtoString := 'Shanghai Fuxu Tech Co., Ltd.';

	16#00688618:
		F_EtherCAT_VendorIDtoString := '3onedata Co., Ltd.';

	16#00688688:
		F_EtherCAT_VendorIDtoString := 'Foshan Augmented Intelligence Technology Co., Ltd.';

	16#00688888:
		F_EtherCAT_VendorIDtoString := 'GUILIN WINDCON CO.,LTD';

	16#00690069:
		F_EtherCAT_VendorIDtoString := 'SHENZHEN HENGKETONG ROBOT CO., LTD';

	16#00691337:
		F_EtherCAT_VendorIDtoString := 'Procada AB';

	16#00696969:
		F_EtherCAT_VendorIDtoString := 'Mianyang Fude Robot Co., Ltd.';

	16#006AFE96:
		F_EtherCAT_VendorIDtoString := 'ShuraCore LLC';

	16#006B4F53:
		F_EtherCAT_VendorIDtoString := 'Kjellberg Finsterwalde Plasma und Maschinen GmbH';

	16#006C6267:
		F_EtherCAT_VendorIDtoString := 'Taiyo Nippon Sanso ATI Corporation';

	16#006D6F74:
		F_EtherCAT_VendorIDtoString := 'motrona GmbH';

	16#006D7361:
		F_EtherCAT_VendorIDtoString := 'Hefei MacroSilicon Technology Co.,Ltd';

	16#006E542D:
		F_EtherCAT_VendorIDtoString := 'Genesis Robotics and Motion Technologies Canada, ULC';

	16#00700000:
		F_EtherCAT_VendorIDtoString := 'TNK CO., LTD.';

	16#00700001:
		F_EtherCAT_VendorIDtoString := 'AE Teknoloji Yazılım Otomasyon Ltd. Şti.';

	16#00700100:
		F_EtherCAT_VendorIDtoString := 'Cyber Control Systems LLC';

	16#00706150:
		F_EtherCAT_VendorIDtoString := 'LogiSolics by Dietmar Steidl';

	16#00706E74:
		F_EtherCAT_VendorIDtoString := 'PONUTech';

	16#007207EC:
		F_EtherCAT_VendorIDtoString := 'Trotec Laser GmbH';

	16#00730220:
		F_EtherCAT_VendorIDtoString := 'PLASOURCE Co., Ltd.';

	16#00737966:
		F_EtherCAT_VendorIDtoString := 'IO Builder Kft.';

	16#00746563:
		F_EtherCAT_VendorIDtoString := 'tecVenture UG (haftungsbeschrankt)';

	16#00746568:
		F_EtherCAT_VendorIDtoString := 'MechAdept Limited';

	16#00746B54:
		F_EtherCAT_VendorIDtoString := 'thyssenkrupp Transrapid GmbH';

	16#00746C65:
		F_EtherCAT_VendorIDtoString := 'BST GmbH';

	16#00750608:
		F_EtherCAT_VendorIDtoString := 'ZHITENG (Shenzhen) Motion Technology Co., Ltd.';

	16#00756500:
		F_EtherCAT_VendorIDtoString := 'Zhuhai Motion Control Motor Co., Ltd.';

	16#00770712:
		F_EtherCAT_VendorIDtoString := 'Rainbow Co.';

	16#00774561:
		F_EtherCAT_VendorIDtoString := 'FLSmidth Ventomatic S.p.A';

	16#0077696E:
		F_EtherCAT_VendorIDtoString := 'krtkl inc.';

	16#00777464:
		F_EtherCAT_VendorIDtoString := 'Wuxi Qasky-comm Quantum Technology Co., LTD';

	16#00777700:
		F_EtherCAT_VendorIDtoString := 'SENTROL Co., Ltd.';

	16#00777777:
		F_EtherCAT_VendorIDtoString := 'HangZhou Dianzi University, School of Mechanical Engineering';

	16#00777ABC:
		F_EtherCAT_VendorIDtoString := 'Industrias Rochin';

	16#00778899:
		F_EtherCAT_VendorIDtoString := 'Shanghai Tianhe Automation Instrumentation Co.,Ltd.';

	16#00779999:
		F_EtherCAT_VendorIDtoString := 'PHUC SON TECHNOLOGY CO., LTD.';

	16#00782782:
		F_EtherCAT_VendorIDtoString := 'Hangzhou Bergerda Automation Technology Co., Ltd.';

	16#00789456:
		F_EtherCAT_VendorIDtoString := 'Devol Advanced Automation, Inc.';

	16#00789789:
		F_EtherCAT_VendorIDtoString := 'Firsttech Design Co., Ltd.';

	16#00796866:
		F_EtherCAT_VendorIDtoString := 'Chengdu Yanxing Automation Engineering Co., Ltd.';

	16#0079796D:
		F_EtherCAT_VendorIDtoString := 'METIS Co., Ltd.';

	16#00799245:
		F_EtherCAT_VendorIDtoString := 'Goldlucke GmbH';

	16#007AFE76:
		F_EtherCAT_VendorIDtoString := 'Promwad Soft LLC';

	16#007DC7DC:
		F_EtherCAT_VendorIDtoString := 'TELE DATA CONTROL, spol. s r. o.';

	16#007E7E7E:
		F_EtherCAT_VendorIDtoString := 'HANGZHOU ZHONGYA MACHINERY CO., LTD.';

	16#00800000:
		F_EtherCAT_VendorIDtoString := 'Shenzhen Hpmont Technology Co., Ltd.';

	16#00800188:
		F_EtherCAT_VendorIDtoString := 'NIDEC READ CORPORATION';

	16#00803804:
		F_EtherCAT_VendorIDtoString := 'Harbin Servo Innovation Technology Co., Ltd';

	16#00811791:
		F_EtherCAT_VendorIDtoString := 'Microtime Computer Inc.';

	16#00811811:
		F_EtherCAT_VendorIDtoString := 'EGICON S.R.L.';

	16#00828845:
		F_EtherCAT_VendorIDtoString := 'AL. Robot Co., Inc.';

	16#00830517:
		F_EtherCAT_VendorIDtoString := 'Korea Institute of Science and Technology (KIST)';

	16#00830518:
		F_EtherCAT_VendorIDtoString := 'Korea Institute of Science and Technology (KIST)';

	16#00830519:
		F_EtherCAT_VendorIDtoString := 'Korea Institute of Science and Technology (KIST)';

	16#00831219:
		F_EtherCAT_VendorIDtoString := 'Chengdu Sino-Tech Smart Energy Co., Ltd.';

	16#00835109:
		F_EtherCAT_VendorIDtoString := 'Ninest Co.,Ltd.';

	16#00836699:
		F_EtherCAT_VendorIDtoString := 'Hunan Aicortech Intelligent Technology Co.,Ltd.';

	16#00850104:
		F_EtherCAT_VendorIDtoString := 'Shenzhen Veichi Electric Co., Ltd';

	16#00850111:
		F_EtherCAT_VendorIDtoString := 'Shenzhen SiCARRIER Technology Co., Ltd.';

	16#00860755:
		F_EtherCAT_VendorIDtoString := 'SHENZHEN STONKER MOTOR CO.,LTD';

	16#00860816:
		F_EtherCAT_VendorIDtoString := 'Sichuan Odot Automation System Co.,Ltd.';

	16#00862413:
		F_EtherCAT_VendorIDtoString := 'REsource Electric Tianjin Ltd.';

	16#00868686:
		F_EtherCAT_VendorIDtoString := 'Changzhou Baolong Motor Co., Ltd.';

	16#00871009:
		F_EtherCAT_VendorIDtoString := 'Suzhou ECMA Industrial Technology Co., Ltd.';

	16#00871217:
		F_EtherCAT_VendorIDtoString := 'Rocket Lab Kft.';

	16#00875111:
		F_EtherCAT_VendorIDtoString := 'Protech Systems Co., Ltd.';

	16#00876543:
		F_EtherCAT_VendorIDtoString := 'KONE Oyj';

	16#00880088:
		F_EtherCAT_VendorIDtoString := 'Atop Technologies, Inc.';

	16#00884443:
		F_EtherCAT_VendorIDtoString := 'Nanjing Solidot Electronic Technology Co., Ltd.';

	16#00884543:
		F_EtherCAT_VendorIDtoString := 'Beijing Mingda Intelligent Control Technology Co., Ltd.';

	16#00886688:
		F_EtherCAT_VendorIDtoString := 'Simplo Technology CO., LTD.';

	16#00888666:
		F_EtherCAT_VendorIDtoString := 'Suzhou Zongwei Technology Co., Ltd.';

	16#00888880:
		F_EtherCAT_VendorIDtoString := 'NINGBO EST TECHNOLOGY CO., LTD';

	16#00888882:
		F_EtherCAT_VendorIDtoString := 'Hitachi High-Technologies Corporation';

	16#00888889:
		F_EtherCAT_VendorIDtoString := 'Shenzhen Hualong Xunda Information Technology Co., Ltd.';

	16#00888999:
		F_EtherCAT_VendorIDtoString := 'Hangzhou Hangtu Technology Co., Ltd.';

	16#00889606:
		F_EtherCAT_VendorIDtoString := 'Dongguan Avatar System Automation Equipment Co., Ltd.';

	16#00889900:
		F_EtherCAT_VendorIDtoString := 'Shanghai Yanlan Automation Technology Co., Ltd.';

	16#00889999:
		F_EtherCAT_VendorIDtoString := 'Hangzhou Wahaha Group Co., LTD., Mechanical and Electrical Institute';

	16#0088F88F:
		F_EtherCAT_VendorIDtoString := 'DaLian Faster Electrical and Mechanical Co., Ltd.';

	16#008C1F64:
		F_EtherCAT_VendorIDtoString := 'TrueNorth Ltd.';

	16#00901146:
		F_EtherCAT_VendorIDtoString := 'Guangdong dingshen Electric Technology Co., Ltd.';

	16#00922189:
		F_EtherCAT_VendorIDtoString := 'Suzhou Quick Laser Technology';

	16#00941136:
		F_EtherCAT_VendorIDtoString := 'Juju Engineering';

	16#00942233:
		F_EtherCAT_VendorIDtoString := 'jhensheng Co.,Ltd.';

	16#00950701:
		F_EtherCAT_VendorIDtoString := 'ULVAC Korea, Ltd.';

	16#00952358:
		F_EtherCAT_VendorIDtoString := 'TROY ENTERPRISE CO., LTD';

	16#00958895:
		F_EtherCAT_VendorIDtoString := 'Beijing Jiyuan Automation Technology Co., Ltd.';

	16#00969696:
		F_EtherCAT_VendorIDtoString := 'GENERTEC HARBIN MEASURING & CUTTING TOOL CO.,LTD.';

	16#00972430:
		F_EtherCAT_VendorIDtoString := 'Moore Nanotechnology Systems, LLC';

	16#00991000:
		F_EtherCAT_VendorIDtoString := 'Shenzhen SuperFar lntelligent Control Technology Co.,LTD.';

	16#00998877:
		F_EtherCAT_VendorIDtoString := 'DATASCHALT engineering GmbH';

	16#00999999:
		F_EtherCAT_VendorIDtoString := 'Smartind Technologies Co., Ltd.';

	16#0099CC66:
		F_EtherCAT_VendorIDtoString := 'WT Microelectronics Co., Ltd.';

	16#0099CF11:
		F_EtherCAT_VendorIDtoString := 'Shenzhen YOOCHIP Electronics Co.,Ltd';

	16#009CFBF1:
		F_EtherCAT_VendorIDtoString := 'MESOMATIC GmbH & Co. KG';

	16#009FA7AC:
		F_EtherCAT_VendorIDtoString := 'Ultima Genomics, Inc.';

	16#00A0000A:
		F_EtherCAT_VendorIDtoString := 'RD2 SRL';

	16#00A0415E:
		F_EtherCAT_VendorIDtoString := 'Opsens Solutions Inc.';

	16#00A12000:
		F_EtherCAT_VendorIDtoString := 'Universitat Politecnica de Valencia, Instituto Universitario de Automatica e Informatica Industrial';

	16#00A1234F:
		F_EtherCAT_VendorIDtoString := 'Shanghai Maritime University, Logistics Engineering College';

	16#00A1BEEF:
		F_EtherCAT_VendorIDtoString := 'F&S PROZESSAUTOMATION GmbH';

	16#00A1C0DE:
		F_EtherCAT_VendorIDtoString := 'Arsenal Engineering S.r.l.';

	16#00A21234:
		F_EtherCAT_VendorIDtoString := 'EMP Designs Ltd';

	16#00A24273:
		F_EtherCAT_VendorIDtoString := 'ASYS Automatic Systems Co., Ltd.';

	16#00A54321:
		F_EtherCAT_VendorIDtoString := 'NEW SOLUTION S.A.';

	16#00A55A5A:
		F_EtherCAT_VendorIDtoString := 'Hikrobot Technology Co., Ltd.';

	16#00A57120:
		F_EtherCAT_VendorIDtoString := 'Venturi Astrolab, Inc.';

	16#00A5C000:
		F_EtherCAT_VendorIDtoString := 'ASC GmbH';

	16#00A5DFF4:
		F_EtherCAT_VendorIDtoString := 'Kenotom P.C.';

	16#00A5E15A:
		F_EtherCAT_VendorIDtoString := 'ASELSAN A.S.';

	16#00A70EA7:
		F_EtherCAT_VendorIDtoString := 'Basemap Inc., DBA Automaton';

	16#00AA0001:
		F_EtherCAT_VendorIDtoString := 'Inventec Appliances (Shanghai) Co., Ltd.';

	16#00AA1314:
		F_EtherCAT_VendorIDtoString := 'HENAN XINZHILIN ELECTROMECHANICAL DEVICE CO.,LTD';

	16#00AA55A5:
		F_EtherCAT_VendorIDtoString := 'Bitvis AS';

	16#00AA55AA:
		F_EtherCAT_VendorIDtoString := 'Shenzhen Sipake Electric Co., Ltd.';

	16#00AA55CF:
		F_EtherCAT_VendorIDtoString := 'Crowtec Bilişim Yazılım Elektronik San. ve Tic. Ltd. Şti';

	16#00AAA111:
		F_EtherCAT_VendorIDtoString := 'Amada Miyachi America, Inc.';

	16#00AAA555:
		F_EtherCAT_VendorIDtoString := 'EMOTIONTEK Co., Ltd.';

	16#00AAAAAA:
		F_EtherCAT_VendorIDtoString := 'Altera Corporation';

	16#00AAAAAD:
		F_EtherCAT_VendorIDtoString := 'Solid Co., LTD.';

	16#00AAAABB:
		F_EtherCAT_VendorIDtoString := 'TDS Technology (S) Pte Ltd.';

	16#00AAABBB:
		F_EtherCAT_VendorIDtoString := 'CRRC QINGDAO SIFANG ROLLING STOCK RESEARCH INSTITUTE Co., Ltd.';

	16#00AACCEE:
		F_EtherCAT_VendorIDtoString := 'Racing Electric Instrument Co., LTD.';

	16#00AAFFAA:
		F_EtherCAT_VendorIDtoString := 'ComSol Inh. Uwe Reinersmann';

	16#00AAFFEE:
		F_EtherCAT_VendorIDtoString := 'High Q Laser GmbH';

	16#00AB0001:
		F_EtherCAT_VendorIDtoString := 'Huizhou Aibo Automatic Control Equipment CO.,LTD.';

	16#00AB12CD:
		F_EtherCAT_VendorIDtoString := 'PyramidTech LLC';

	16#00AB1AB1:
		F_EtherCAT_VendorIDtoString := 'ABIMAN ENGINEERING CO., LTD';

	16#00AB24FC:
		F_EtherCAT_VendorIDtoString := 'NovaTech LLC';

	16#00ABA000:
		F_EtherCAT_VendorIDtoString := 'abaxor engineering GmbH';

	16#00ABA1EC:
		F_EtherCAT_VendorIDtoString := 'abatec group ag';

	16#00ABAB00:
		F_EtherCAT_VendorIDtoString := 'Pearls of Life AB';

	16#00ABF159:
		F_EtherCAT_VendorIDtoString := 'Promotion Comercio e Servico Ltda';

	16#00ACCE55:
		F_EtherCAT_VendorIDtoString := 'enders GmbH';

	16#00ACDCAB:
		F_EtherCAT_VendorIDtoString := 'Siemens Gamesa Renewable Energy A/S';

	16#00ACDCAC:
		F_EtherCAT_VendorIDtoString := 'Siemens Gamesa Renewable Energy Ltd';

	16#00ACEACE:
		F_EtherCAT_VendorIDtoString := 'HANYANG ROBOTICS CO.,LTD';

	16#00ADCAFE:
		F_EtherCAT_VendorIDtoString := 'Analog Devices, Inc.';

	16#00AE4B4B:
		F_EtherCAT_VendorIDtoString := 'KK Wind Solutions A/S';

	16#00AE86FD:
		F_EtherCAT_VendorIDtoString := 'HOFO Automation Co., Ltd.';

	16#00AEA000:
		F_EtherCAT_VendorIDtoString := 'AEA Srl';

	16#00AF2497:
		F_EtherCAT_VendorIDtoString := 'Yeungnam University, College of Mechanical and IT Engineering, Department of Information and Communication Engineering, Advanced Networking Technology Lab.';

	16#00B071C5:
		F_EtherCAT_VendorIDtoString := 'PAL Robotics S.L.';

	16#00B07B07:
		F_EtherCAT_VendorIDtoString := 'Remedy Robotics, Inc.';

	16#00B100D5:
		F_EtherCAT_VendorIDtoString := 'King’s College London, Faculty of Life Sciences & Medicine, School of Biomedical Engineering & Imaging Sciences';

	16#00B12B12:
		F_EtherCAT_VendorIDtoString := 'Jingxin Plasma Technology Co.Ltd.';

	16#00B7AD11:
		F_EtherCAT_VendorIDtoString := 'Tecnomatic SA';

	16#00BA5E20:
		F_EtherCAT_VendorIDtoString := 'Hangzhou Xieneng Technology Co., Ltd.';

	16#00BABE42:
		F_EtherCAT_VendorIDtoString := 'UCY Technologies GmbH';

	16#00BADA55:
		F_EtherCAT_VendorIDtoString := 'NEWTEC A/S';

	16#00BADBEE:
		F_EtherCAT_VendorIDtoString := '4NXT S.r.l.';

	16#00BADFAB:
		F_EtherCAT_VendorIDtoString := 'KNDS France S.A.';

	16#00BAFF1E:
		F_EtherCAT_VendorIDtoString := 'Memjet Technology Ltd';

	16#00BBBBBB:
		F_EtherCAT_VendorIDtoString := 'BLUESINK Co., Ltd';

	16#00BEE000:
		F_EtherCAT_VendorIDtoString := 'm-Bee GmbH';

	16#00BF0001:
		F_EtherCAT_VendorIDtoString := 'Be-Friend Technology Inc.';

	16#00C007D9:
		F_EtherCAT_VendorIDtoString := 'Guangdong Coordy Numerical Control Technology Co.,Ltd.';

	16#00C0DE20:
		F_EtherCAT_VendorIDtoString := 'Martec Engineering GmbH';

	16#00C0FFEE:
		F_EtherCAT_VendorIDtoString := 'Moog Animatics';

	16#00C57C57:
		F_EtherCAT_VendorIDtoString := 'Chemspeed Technologies AG';

	16#00CA13F1:
		F_EtherCAT_VendorIDtoString := 'Canon Production Printing Netherlands B.V.';

	16#00CA13F2:
		F_EtherCAT_VendorIDtoString := 'Canon Production Printing Germany GmbH & Co. KG';

	16#00CA71EB:
		F_EtherCAT_VendorIDtoString := 'SENER Aeroespacial, S.A.';

	16#00CABEAD:
		F_EtherCAT_VendorIDtoString := 'Kyland Technology Co., Ltd.';

	16#00CADCAD:
		F_EtherCAT_VendorIDtoString := 'IML Co. Ltd.';

	16#00CC00AA:
		F_EtherCAT_VendorIDtoString := 'Saenggaksaemteo Co.';

	16#00CC1982:
		F_EtherCAT_VendorIDtoString := 'Comtrol Corporation';

	16#00CCCCCC:
		F_EtherCAT_VendorIDtoString := 'Largan Precision Co.,Ltd.';

	16#00CDCDAB:
		F_EtherCAT_VendorIDtoString := 'Hanwha Aerospace Co., Ltd.';

	16#00CE7C21:
		F_EtherCAT_VendorIDtoString := 'China Electronics Technology Group Corporation No. 21 Research Institute';

	16#00CECECE:
		F_EtherCAT_VendorIDtoString := 'Canon Electronics Inc.';

	16#00D02379:
		F_EtherCAT_VendorIDtoString := 'REXA Inc.';

	16#00D2EA3E:
		F_EtherCAT_VendorIDtoString := 'Dreame Innovation Technology (Suzhou) Co., Ltd.';

	16#00D56130:
		F_EtherCAT_VendorIDtoString := 'Lowenstein Medical GmbH & Co. KG';

	16#00D87688:
		F_EtherCAT_VendorIDtoString := 'Robo Biz Core Co., Ltd';

	16#00DA4E00:
		F_EtherCAT_VendorIDtoString := 'DAVE Srl';

	16#00DAD001:
		F_EtherCAT_VendorIDtoString := 'Studio elektronike Rijeka d.o.o.';

	16#00DAEAC0:
		F_EtherCAT_VendorIDtoString := 'DAEATI Co., Ltd.';

	16#00DCAC88:
		F_EtherCAT_VendorIDtoString := 'Le-AutomatiX (Shanghai) Co., Ltd.';

	16#00DDDDDD:
		F_EtherCAT_VendorIDtoString := 'DAINCUBE INC.';

	16#00DEADBF:
		F_EtherCAT_VendorIDtoString := 'Shanghai xPartner Robotics Co.,Ltd.';

	16#00DECADE:
		F_EtherCAT_VendorIDtoString := 'Insoptics Sp. z O.O.';

	16#00DEDBEF:
		F_EtherCAT_VendorIDtoString := 'Dexterity, Inc.';

	16#00DFE603:
		F_EtherCAT_VendorIDtoString := 'Dover Flexo Electronics, Inc.';

	16#00E05DA6:
		F_EtherCAT_VendorIDtoString := 'Detlef Fink Elektronik-& Softwareentwicklung';

	16#00E11FE1:
		F_EtherCAT_VendorIDtoString := 'Elife International S.r.l.';

	16#00E50E50:
		F_EtherCAT_VendorIDtoString := 'ESO, European Southern Observatory';

	16#00E57AB1:
		F_EtherCAT_VendorIDtoString := 'Estabili Tecnologia';

	16#00E5CA18:
		F_EtherCAT_VendorIDtoString := 'Weld Tooling Corporation (dba BUG-O Systems)';

	16#00EA7506:
		F_EtherCAT_VendorIDtoString := 'Shanghai Gaviota Intelligent Technology Co., Ltd.';

	16#00EA8888:
		F_EtherCAT_VendorIDtoString := 'Shenzhen Evta Technology Co., Ltd.';

	16#00EAEB01:
		F_EtherCAT_VendorIDtoString := 'NetEase (Hangzhou) Network Co., Ltd.';

	16#00EC1608:
		F_EtherCAT_VendorIDtoString := 'Tongtai Machine & Tool Co., Ltd.';

	16#00EC1991:
		F_EtherCAT_VendorIDtoString := 'PROMAX srl';

	16#00EC2018:
		F_EtherCAT_VendorIDtoString := 'PRODRIVES & MOTIONS CO., LTD.';

	16#00EC4800:
		F_EtherCAT_VendorIDtoString := 'Hitex (UK) Ltd.';

	16#00EC8888:
		F_EtherCAT_VendorIDtoString := 'E-Champion Laser Tech (Jiangsu) Co., Ltd.';

	16#00ECADC0:
		F_EtherCAT_VendorIDtoString := 'Encoder Products Company';

	16#00ECADE1:
		F_EtherCAT_VendorIDtoString := 'Mecademic Inc.';

	16#00ECEEDA:
		F_EtherCAT_VendorIDtoString := 'Exceed Automation, LLC';

	16#00EDA168:
		F_EtherCAT_VendorIDtoString := 'Endex Automation Technology Co., Ltd.';

	16#00EDC0DE:
		F_EtherCAT_VendorIDtoString := 'STOGRA Antriebstechnik GmbH';

	16#00EE00AA:
		F_EtherCAT_VendorIDtoString := 'ENTEC Electric & Electronic CO., LTD.';

	16#00EE1000:
		F_EtherCAT_VendorIDtoString := 'Euto Energy Elektronik San. ve Tic. Ltd. Sti.';

	16#00EECCAA:
		F_EtherCAT_VendorIDtoString := 'Beijing Aurasky Electronics Co., Ltd.';

	16#00EEE669:
		F_EtherCAT_VendorIDtoString := 'Henan Mechanical and Electrical Vocational College';

	16#00EEEEEE:
		F_EtherCAT_VendorIDtoString := 'Swyss Electronics GmbH';

	16#00F0AE1B:
		F_EtherCAT_VendorIDtoString := 'NTCSOFT Co., Ltd.';

	16#00F1CA42:
		F_EtherCAT_VendorIDtoString := 'Meccanica 42 S.r.l.';

	16#00F1F1F1:
		F_EtherCAT_VendorIDtoString := 'Williams Grand Prix Engineering Limited';

	16#00F2020F:
		F_EtherCAT_VendorIDtoString := 'MİLTEKSAN CNC Teknoloji ve Kontrol Sistemleri Sanayi A.Ş.';

	16#00F2F2F2:
		F_EtherCAT_VendorIDtoString := 'spectral process Ingenieurburo';

	16#00F5CB27:
		F_EtherCAT_VendorIDtoString := 'Alpha Project Co.,Ltd.';

	16#00F8F8F8:
		F_EtherCAT_VendorIDtoString := 'Suzhou Otronic Medical Technology Co., Ltd.';

	16#00FA1337:
		F_EtherCAT_VendorIDtoString := 'British Columbia Institute of Technology';

	16#00FA140A:
		F_EtherCAT_VendorIDtoString := 'JTEKT ELECTRONICS CORPORATION';

	16#00FA3C77:
		F_EtherCAT_VendorIDtoString := 'DNV Electronics, LLC';

	16#00FABADA:
		F_EtherCAT_VendorIDtoString := 'GTD Sistemas de Informacion SA';

	16#00FC37A4:
		F_EtherCAT_VendorIDtoString := 'Hirocon Corporation';

	16#00FDC42D:
		F_EtherCAT_VendorIDtoString := 'MECOS AG';

	16#00FE0001:
		F_EtherCAT_VendorIDtoString := 'Kemppi Oy';

	16#00FEDABC:
		F_EtherCAT_VendorIDtoString := 'Mouvent AG';

	16#00FEDCAB:
		F_EtherCAT_VendorIDtoString := 'Shanghai Shaoyu Automation Design Co., Ltd.';

	16#00FEDCBA:
		F_EtherCAT_VendorIDtoString := 'E-TEAM di Righini Bruno & C. S.a.s.';

	16#00FF00AA:
		F_EtherCAT_VendorIDtoString := 'Dongguan Precision Intelligent Technology Co., Ltd.';

	16#00FF00F0:
		F_EtherCAT_VendorIDtoString := 'Eagle Technologies';

	16#00FF00FF:
		F_EtherCAT_VendorIDtoString := 'TDK-Lambda Ltd.';

	16#00FF2000:
		F_EtherCAT_VendorIDtoString := 'Hangzhou Seenpin Electromechanical Transmission Co., Ltd.';

	16#00FF88FF:
		F_EtherCAT_VendorIDtoString := 'Beijing Information Science & Technology University, School of Instrument Science and Opto-Electronics Engineering';

	16#00FFAABB:
		F_EtherCAT_VendorIDtoString := 'YOSIO ELECTRONIC COMPANY';

	16#00FFF888:
		F_EtherCAT_VendorIDtoString := 'UTEK TECHNOLOGY (SHENZHEN) CO., LTD.';

	16#00FFFAAA:
		F_EtherCAT_VendorIDtoString := 'Xiamen Zhengai Technology Co., Ltd.';

	16#00FFFF22:
		F_EtherCAT_VendorIDtoString := 'Anhui LAEG Electric Co., Ltd';

	16#00FFFFFF:
		F_EtherCAT_VendorIDtoString := 'Chongqing Huashu Robotics Co.,Ltd.';

	16#01000001:
		F_EtherCAT_VendorIDtoString := 'Arlington Laboratory Corporation';

